LIN {X 0,Y 496.711,Z 403.86,A -85,B 0,C 180,E1 23580.115,E2 23580.115} C_VEL
LIN {X 0,Y 496.741,Z 403.852,A -85,B 0,C 180,E1 23576.65,E2 23576.65} C_VEL
LIN {X 0,Y 496.767,Z 403.854,A -85,B 0,C 180,E1 23573.18,E2 23573.18} C_VEL
LIN {X 0,Y 496.731,Z 403.861,A -85,B 0,C 180,E1 23569.68,E2 23569.68} C_VEL
LIN {X 0,Y 496.739,Z 403.856,A -85,B 0,C 180,E1 23566.141,E2 23566.141} C_VEL
LIN {X 0,Y 496.771,Z 403.853,A -85,B 0,C 180,E1 23562.669,E2 23562.669} C_VEL
LIN {X 0,Y 496.766,Z 403.847,A -85,B 0,C 180,E1 23559.041,E2 23559.041} C_VEL
LIN {X 0,Y 496.807,Z 404.124,A -85,B 0,C 180,E1 23556.819,E2 23556.819} C_VEL
LIN {X 0,Y 499.675,Z 411.051,A -85,B 0,C 180,E1 23555.782,E2 23555.782} C_VEL
LIN {X 0,Y 507.249,Z 429.235,A -85,B 0,C 180,E1 23553.293,E2 23553.293} C_VEL
LIN {X 0,Y 509.58,Z 435.728,A -85,B 0,C 180,E1 23552.475,E2 23552.475} C_VEL
LIN {X 0,Y 508.606,Z 453.094,A -85,B 0,C 180,E1 23551.014,E2 23551.014} C_VEL
LIN {X 0,Y 512.123,Z 472.591,A -85,B 0,C 180,E1 23550.372,E2 23550.372} C_VEL
LIN {X 0,Y 509.75,Z 617.433,A -85,B 0,C 180,E1 23548.089,E2 23548.089} C_VEL
LIN {X 0,Y 508.797,Z 625.124,A -85,B 0,C 180,E1 23548.03,E2 23548.03} C_VEL
LIN {X 0,Y 503.244,Z 645.629,A -85,B 0,C 180,E1 23548.096,E2 23548.096} C_VEL
LIN {X 0,Y 502.511,Z 652.229,A -85,B 0,C 180,E1 23548.038,E2 23548.038} C_VEL
LIN {X 0,Y 501.351,Z 717.097,A -85,B 0,C 180,E1 23546.975,E2 23546.975} C_VEL
LIN {X 0,Y 500.539,Z 738.052,A -85,B 0,C 180,E1 23546.417,E2 23546.417} C_VEL
LIN {X 0,Y 499.534,Z 757.461,A -85,B 0,C 180,E1 23545.684,E2 23545.684} C_VEL
LIN {X 0,Y 498.294,Z 776.687,A -85,B 0,C 180,E1 23544.746,E2 23544.746} C_VEL
LIN {X 0,Y 496.904,Z 795.621,A -85,B 0,C 180,E1 23543.587,E2 23543.587} C_VEL
LIN {X 0,Y 495.479,Z 813.178,A -85,B 0,C 180,E1 23542.277,E2 23542.277} C_VEL
LIN {X 0,Y 494.06,Z 829.63,A -85,B 0,C 180,E1 23540.808,E2 23540.808} C_VEL
LIN {X 0,Y 492.634,Z 845.536,A -85,B 0,C 180,E1 23539.11,E2 23539.11} C_VEL
LIN {X 0,Y 491.345,Z 860.076,A -85,B 0,C 180,E1 23537.269,E2 23537.269} C_VEL
LIN {X 0,Y 490.236,Z 873.347,A -85,B 0,C 180,E1 23535.28,E2 23535.28} C_VEL
LIN {X 0,Y 489.325,Z 886.414,A -85,B 0,C 180,E1 23532.986,E2 23532.986} C_VEL
LIN {X 0,Y 488.72,Z 897.123,A -85,B 0,C 180,E1 23530.736,E2 23530.736} C_VEL
LIN {X 0,Y 488.32,Z 905.885,A -85,B 0,C 180,E1 23528.491,E2 23528.491} C_VEL
LIN {X 0,Y 488.079,Z 913.183,A -85,B 0,C 180,E1 23526.152,E2 23526.152} C_VEL
LIN {X 0,Y 487.966,Z 918.575,A -85,B 0,C 180,E1 23523.868,E2 23523.868} C_VEL
LIN {X 0,Y 487.921,Z 922.481,A -85,B 0,C 180,E1 23521.499,E2 23521.499} C_VEL
LIN {X 0,Y 487.912,Z 924.811,A -85,B 0,C 180,E1 23519.053,E2 23519.053} C_VEL
LIN {X 0,Y 487.907,Z 925.448,A -85,B 0,C 180,E1 23516.662,E2 23516.662} C_VEL
LIN {X 0,Y 487.911,Z 924.503,A -85,B 0,C 180,E1 23514.321,E2 23514.321} C_VEL
LIN {X 0,Y 487.927,Z 921.952,A -85,B 0,C 180,E1 23512.021,E2 23512.021} C_VEL
LIN {X 0,Y 487.973,Z 917.691,A -85,B 0,C 180,E1 23509.632,E2 23509.632} C_VEL
LIN {X 0,Y 488.118,Z 911.798,A -85,B 0,C 180,E1 23507.275,E2 23507.275} C_VEL
LIN {X 0,Y 488.374,Z 904.684,A -85,B 0,C 180,E1 23505.068,E2 23505.068} C_VEL
LIN {X 0,Y 488.809,Z 895.342,A -85,B 0,C 180,E1 23502.76,E2 23502.76} C_VEL
LIN {X 0,Y 489.437,Z 884.661,A -85,B 0,C 180,E1 23500.592,E2 23500.592} C_VEL
LIN {X 0,Y 490.443,Z 870.664,A -85,B 0,C 180,E1 23498.202,E2 23498.202} C_VEL
LIN {X 0,Y 491.534,Z 857.477,A -85,B 0,C 180,E1 23496.304,E2 23496.304} C_VEL
LIN {X 0,Y 492.839,Z 842.493,A -85,B 0,C 180,E1 23494.477,E2 23494.477} C_VEL
LIN {X 0,Y 494.246,Z 826.553,A -85,B 0,C 180,E1 23492.838,E2 23492.838} C_VEL
LIN {X 0,Y 495.672,Z 809.764,A -85,B 0,C 180,E1 23491.385,E2 23491.385} C_VEL
LIN {X 0,Y 497.08,Z 792.089,A -85,B 0,C 180,E1 23490.113,E2 23490.113} C_VEL
LIN {X 0,Y 498.389,Z 773.462,A -85,B 0,C 180,E1 23489.02,E2 23489.02} C_VEL
LIN {X 0,Y 499.54,Z 754.515,A -85,B 0,C 180,E1 23488.134,E2 23488.134} C_VEL
LIN {X 0,Y 500.549,Z 733.899,A -85,B 0,C 180,E1 23487.4,E2 23487.4} C_VEL
LIN {X 0,Y 501.274,Z 713.46,A -85,B 0,C 180,E1 23486.893,E2 23486.893} C_VEL
LIN {X 0,Y 505.137,Z 479.595,A -85,B 0,C 180,E1 23483.179,E2 23483.179} C_VEL
LIN {X 0,Y 505.027,Z 471.969,A -85,B 0,C 180,E1 23483.036,E2 23483.036} C_VEL
LIN {X 0,Y 501.4,Z 452.019,A -85,B 0,C 180,E1 23482.346,E2 23482.346} C_VEL
LIN {X 0,Y 502.149,Z 437.999,A -85,B 0,C 180,E1 23481.121,E2 23481.121} C_VEL
LIN {X 0,Y 494.668,Z 418.979,A -85,B 0,C 180,E1 23478.615,E2 23478.615} C_VEL
LIN {X 0,Y 488.848,Z 405.013,A -85,B 0,C 180,E1 23476.605,E2 23476.605} C_VEL
LIN {X 0,Y 488.821,Z 404.811,A -85,B 0,C 180,E1 23472.99,E2 23472.99} C_VEL
LIN {X 0,Y 488.827,Z 404.843,A -85,B 0,C 180,E1 23469.4,E2 23469.4} C_VEL
LIN {X 0,Y 488.81,Z 404.825,A -85,B 0,C 180,E1 23465.825,E2 23465.825} C_VEL
LIN {X 0,Y 488.828,Z 404.838,A -85,B 0,C 180,E1 23462.333,E2 23462.333} C_VEL
LIN {X 0,Y 488.826,Z 404.833,A -85,B 0,C 180,E1 23458.697,E2 23458.697} C_VEL
LIN {X 0,Y 488.816,Z 404.833,A -85,B 0,C 180,E1 23455.109,E2 23455.109} C_VEL
LIN {X 0,Y 488.818,Z 404.835,A -85,B 0,C 180,E1 23451.549,E2 23451.549} C_VEL
LIN {X 0,Y 488.823,Z 404.846,A -85,B 0,C 180,E1 23448.019,E2 23448.019} C_VEL
LIN {X 0,Y 488.827,Z 404.84,A -85,B 0,C 180,E1 23444.39,E2 23444.39} C_VEL
LIN {X 0,Y 488.815,Z 404.84,A -85,B 0,C 180,E1 23440.813,E2 23440.813} C_VEL
LIN {X 0,Y 488.824,Z 404.834,A -85,B 0,C 180,E1 23437.262,E2 23437.262} C_VEL
LIN {X 0,Y 488.82,Z 404.845,A -85,B 0,C 180,E1 23433.642,E2 23433.642} C_VEL
LIN {X 0,Y 488.832,Z 404.835,A -85,B 0,C 180,E1 23430.075,E2 23430.075} C_VEL
LIN {X 0,Y 488.817,Z 404.83,A -85,B 0,C 180,E1 23426.482,E2 23426.482} C_VEL
LIN {X 0,Y 488.829,Z 404.846,A -85,B 0,C 180,E1 23422.87,E2 23422.87} C_VEL
LIN {X 0,Y 488.818,Z 404.831,A -85,B 0,C 180,E1 23419.228,E2 23419.228} C_VEL
LIN {X 0,Y 488.826,Z 404.834,A -85,B 0,C 180,E1 23415.664,E2 23415.664} C_VEL
LIN {X 0,Y 488.82,Z 404.846,A -85,B 0,C 180,E1 23412.043,E2 23412.043} C_VEL
LIN {X 0,Y 488.822,Z 404.831,A -85,B 0,C 180,E1 23408.469,E2 23408.469} C_VEL
LIN {X 0,Y 488.818,Z 404.841,A -85,B 0,C 180,E1 23404.811,E2 23404.811} C_VEL
LIN {X 0,Y 488.827,Z 404.84,A -85,B 0,C 180,E1 23401.172,E2 23401.172} C_VEL
LIN {X 0,Y 488.821,Z 404.834,A -85,B 0,C 180,E1 23397.538,E2 23397.538} C_VEL
LIN {X 0,Y 488.82,Z 404.843,A -85,B 0,C 180,E1 23394.012,E2 23394.012} C_VEL
LIN {X 0,Y 488.817,Z 404.843,A -85,B 0,C 180,E1 23390.345,E2 23390.345} C_VEL
LIN {X 0,Y 488.827,Z 404.84,A -85,B 0,C 180,E1 23386.757,E2 23386.757} C_VEL
LIN {X 0,Y 488.823,Z 404.836,A -85,B 0,C 180,E1 23383.115,E2 23383.115} C_VEL
LIN {X 0,Y 488.817,Z 404.839,A -85,B 0,C 180,E1 23379.527,E2 23379.527} C_VEL
LIN {X 0,Y 488.814,Z 404.842,A -85,B 0,C 180,E1 23375.852,E2 23375.852} C_VEL
LIN {X 0,Y 488.827,Z 404.839,A -85,B 0,C 180,E1 23372.335,E2 23372.335} C_VEL
LIN {X 0,Y 488.829,Z 404.839,A -85,B 0,C 180,E1 23368.699,E2 23368.699} C_VEL
LIN {X 0,Y 488.812,Z 404.84,A -85,B 0,C 180,E1 23365.111,E2 23365.111} C_VEL
LIN {X 0,Y 488.823,Z 404.841,A -85,B 0,C 180,E1 23361.552,E2 23361.552} C_VEL
LIN {X 0,Y 488.824,Z 404.846,A -85,B 0,C 180,E1 23358.021,E2 23358.021} C_VEL
LIN {X 0,Y 488.862,Z 405.087,A -85,B 0,C 180,E1 23355.482,E2 23355.482} C_VEL
LIN {X 0,Y 489.862,Z 407.901,A -85,B 0,C 180,E1 23355.072,E2 23355.072} C_VEL
LIN {X 0,Y 496.792,Z 422.284,A -85,B 0,C 180,E1 23353.182,E2 23353.182} C_VEL
LIN {X 0,Y 506.367,Z 443.634,A -85,B 0,C 180,E1 23350.626,E2 23350.626} C_VEL
LIN {X 0,Y 505.843,Z 455.638,A -85,B 0,C 180,E1 23349.815,E2 23349.815} C_VEL
LIN {X 0,Y 509.16,Z 477.639,A -85,B 0,C 180,E1 23349.149,E2 23349.149} C_VEL
LIN {X 0,Y 505.882,Z 697.396,A -85,B 0,C 180,E1 23345.689,E2 23345.689} C_VEL
LIN {X 0,Y 504.837,Z 762.385,A -85,B 0,C 180,E1 23344.65,E2 23344.65} C_VEL
LIN {X 0,Y 503.952,Z 783.667,A -85,B 0,C 180,E1 23344.113,E2 23344.113} C_VEL
LIN {X 0,Y 502.769,Z 806.1,A -85,B 0,C 180,E1 23343.331,E2 23343.331} C_VEL
LIN {X 0,Y 501.542,Z 826.208,A -85,B 0,C 180,E1 23342.432,E2 23342.432} C_VEL
LIN {X 0,Y 500.044,Z 845.015,A -85,B 0,C 180,E1 23341.373,E2 23341.373} C_VEL
LIN {X 0,Y 498.311,Z 865.469,A -85,B 0,C 180,E1 23339.976,E2 23339.976} C_VEL
LIN {X 0,Y 496.647,Z 883.732,A -85,B 0,C 180,E1 23338.5,E2 23338.5} C_VEL
LIN {X 0,Y 494.933,Z 901.867,A -85,B 0,C 180,E1 23336.758,E2 23336.758} C_VEL
LIN {X 0,Y 493.329,Z 918.653,A -85,B 0,C 180,E1 23334.871,E2 23334.871} C_VEL
LIN {X 0,Y 491.921,Z 934.162,A -85,B 0,C 180,E1 23332.846,E2 23332.846} C_VEL
LIN {X 0,Y 490.71,Z 948.618,A -85,B 0,C 180,E1 23330.642,E2 23330.642} C_VEL
LIN {X 0,Y 489.723,Z 961.442,A -85,B 0,C 180,E1 23328.328,E2 23328.328} C_VEL
LIN {X 0,Y 488.985,Z 972.802,A -85,B 0,C 180,E1 23325.904,E2 23325.904} C_VEL
LIN {X 0,Y 488.492,Z 982.252,A -85,B 0,C 180,E1 23323.496,E2 23323.496} C_VEL
LIN {X 0,Y 488.184,Z 989.875,A -85,B 0,C 180,E1 23321.102,E2 23321.102} C_VEL
LIN {X 0,Y 488.014,Z 996.141,A -85,B 0,C 180,E1 23318.604,E2 23318.604} C_VEL
LIN {X 0,Y 487.94,Z 1000.819,A -85,B 0,C 180,E1 23316.119,E2 23316.119} C_VEL
LIN {X 0,Y 487.912,Z 1003.791,A -85,B 0,C 180,E1 23313.639,E2 23313.639} C_VEL
LIN {X 0,Y 487.908,Z 1005.304,A -85,B 0,C 180,E1 23311.059,E2 23311.059} C_VEL
LIN {X 0,Y 487.907,Z 1005.259,A -85,B 0,C 180,E1 23308.711,E2 23308.711} C_VEL
LIN {X 0,Y 487.91,Z 1003.674,A -85,B 0,C 180,E1 23306.243,E2 23306.243} C_VEL
LIN {X 0,Y 487.944,Z 1000.637,A -85,B 0,C 180,E1 23303.768,E2 23303.768} C_VEL
LIN {X 0,Y 488.018,Z 995.896,A -85,B 0,C 180,E1 23301.282,E2 23301.282} C_VEL
LIN {X 0,Y 488.206,Z 989.183,A -85,B 0,C 180,E1 23298.664,E2 23298.664} C_VEL
LIN {X 0,Y 488.532,Z 981.438,A -85,B 0,C 180,E1 23296.269,E2 23296.269} C_VEL
LIN {X 0,Y 489.045,Z 971.794,A -85,B 0,C 180,E1 23293.859,E2 23293.859} C_VEL
LIN {X 0,Y 489.807,Z 960.2,A -85,B 0,C 180,E1 23291.434,E2 23291.434} C_VEL
LIN {X 0,Y 490.765,Z 947.883,A -85,B 0,C 180,E1 23289.241,E2 23289.241} C_VEL
LIN {X 0,Y 491.917,Z 934.198,A -85,B 0,C 180,E1 23287.16,E2 23287.16} C_VEL
LIN {X 0,Y 493.326,Z 918.696,A -85,B 0,C 180,E1 23285.134,E2 23285.134} C_VEL
LIN {X 0,Y 494.944,Z 901.731,A -85,B 0,C 180,E1 23283.228,E2 23283.228} C_VEL
LIN {X 0,Y 496.642,Z 883.791,A -85,B 0,C 180,E1 23281.505,E2 23281.505} C_VEL
LIN {X 0,Y 498.306,Z 865.543,A -85,B 0,C 180,E1 23280.029,E2 23280.029} C_VEL
LIN {X 0,Y 500.043,Z 845.02,A -85,B 0,C 180,E1 23278.627,E2 23278.627} C_VEL
LIN {X 0,Y 501.533,Z 826.304,A -85,B 0,C 180,E1 23277.573,E2 23277.573} C_VEL
LIN {X 0,Y 502.801,Z 805.216,A -85,B 0,C 180,E1 23276.636,E2 23276.636} C_VEL
LIN {X 0,Y 503.96,Z 782.783,A -85,B 0,C 180,E1 23275.868,E2 23275.868} C_VEL
LIN {X 0,Y 504.819,Z 761.32,A -85,B 0,C 180,E1 23275.337,E2 23275.337} C_VEL
LIN {X 0,Y 506.726,Z 630.415,A -85,B 0,C 180,E1 23273.284,E2 23273.284} C_VEL
LIN {X 0,Y 508.834,Z 475.555,A -85,B 0,C 180,E1 23270.839,E2 23270.839} C_VEL
LIN {X 0,Y 505.533,Z 454.855,A -85,B 0,C 180,E1 23270.2,E2 23270.2} C_VEL
LIN {X 0,Y 506.097,Z 443.386,A -85,B 0,C 180,E1 23269.404,E2 23269.404} C_VEL
LIN {X 0,Y 495.503,Z 419.708,A -85,B 0,C 180,E1 23266.588,E2 23266.588} C_VEL
LIN {X 0,Y 490.039,Z 408.23,A -85,B 0,C 180,E1 23265.072,E2 23265.072} C_VEL
LIN {X 0,Y 488.851,Z 405.059,A -85,B 0,C 180,E1 23264.596,E2 23264.596} C_VEL
LIN {X 0,Y 488.793,Z 404.851,A -85,B 0,C 180,E1 23261.175,E2 23261.175} C_VEL
LIN {X 0,Y 488.817,Z 404.848,A -85,B 0,C 180,E1 23257.672,E2 23257.672} C_VEL
LIN {X 0,Y 488.825,Z 404.842,A -85,B 0,C 180,E1 23254.086,E2 23254.086} C_VEL
LIN {X 0,Y 488.781,Z 404.849,A -85,B 0,C 180,E1 23250.621,E2 23250.621} C_VEL
LIN {X 0,Y 488.772,Z 404.844,A -85,B 0,C 180,E1 23247.009,E2 23247.009} C_VEL
LIN {X 0,Y 488.826,Z 404.841,A -85,B 0,C 180,E1 23243.612,E2 23243.612} C_VEL
LIN {X 0,Y 488.769,Z 404.846,A -85,B 0,C 180,E1 23240.225,E2 23240.225} C_VEL
LIN {X 0,Y 488.751,Z 404.852,A -85,B 0,C 180,E1 23236.642,E2 23236.642} C_VEL
LIN {X 0,Y 488.795,Z 404.851,A -85,B 0,C 180,E1 23233.244,E2 23233.244} C_VEL
LIN {X 0,Y 488.782,Z 404.851,A -85,B 0,C 180,E1 23229.775,E2 23229.775} C_VEL
LIN {X 0,Y 488.76,Z 404.85,A -85,B 0,C 180,E1 23226.342,E2 23226.342} C_VEL
LIN {X 0,Y 488.806,Z 404.843,A -85,B 0,C 180,E1 23222.931,E2 23222.931} C_VEL
LIN {X 0,Y 488.801,Z 404.846,A -85,B 0,C 180,E1 23219.531,E2 23219.531} C_VEL
LIN {X 0,Y 488.778,Z 404.842,A -85,B 0,C 180,E1 23216.011,E2 23216.011} C_VEL
LIN {X 0,Y 488.804,Z 404.847,A -85,B 0,C 180,E1 23212.477,E2 23212.477} C_VEL
LIN {X 0,Y 488.833,Z 404.841,A -85,B 0,C 180,E1 23208.915,E2 23208.915} C_VEL
LIN {X 0,Y 488.813,Z 404.849,A -85,B 0,C 180,E1 23205.307,E2 23205.307} C_VEL
LIN {X 0,Y 488.8,Z 404.848,A -85,B 0,C 180,E1 23201.761,E2 23201.761} C_VEL
LIN {X 0,Y 488.826,Z 404.827,A -85,B 0,C 180,E1 23198.21,E2 23198.21} C_VEL
LIN {X 0,Y 488.87,Z 405.268,A -85,B 0,C 180,E1 23197.562,E2 23197.562} C_VEL
LIN {X 0,Y 496.721,Z 423.489,A -85,B 0,C 180,E1 23194.866,E2 23194.866} C_VEL
LIN {X 0,Y 502.751,Z 438.85,A -85,B 0,C 180,E1 23192.811,E2 23192.811} C_VEL
LIN {X 0,Y 501.912,Z 453.11,A -85,B 0,C 180,E1 23191.6,E2 23191.6} C_VEL
LIN {X 0,Y 505.677,Z 473.944,A -85,B 0,C 180,E1 23190.891,E2 23190.891} C_VEL
LIN {X 0,Y 502.511,Z 652.229,A -85,B 0,C 180,E1 23188.038,E2 23188.038} C_VEL
LIN {X 0,Y 501.556,Z 659.917,A -85,B 0,C 180,E1 23187.978,E2 23187.978} C_VEL
LIN {X 0,Y 495.97,Z 680.411,A -85,B 0,C 180,E1 23188.046,E2 23188.046} C_VEL
LIN {X 0,Y 495.215,Z 687.011,A -85,B 0,C 180,E1 23187.989,E2 23187.989} C_VEL
LIN {X 0,Y 494.51,Z 719.382,A -85,B 0,C 180,E1 23187.421,E2 23187.421} C_VEL
LIN {X 0,Y 493.662,Z 739.881,A -85,B 0,C 180,E1 23186.854,E2 23186.854} C_VEL
LIN {X 0,Y 492.59,Z 759.03,A -85,B 0,C 180,E1 23186.111,E2 23186.111} C_VEL
LIN {X 0,Y 491.254,Z 778.214,A -85,B 0,C 180,E1 23185.151,E2 23185.151} C_VEL
LIN {X 0,Y 489.725,Z 797.454,A -85,B 0,C 180,E1 23183.943,E2 23183.943} C_VEL
LIN {X 0,Y 488.108,Z 815.828,A -85,B 0,C 180,E1 23182.527,E2 23182.527} C_VEL
LIN {X 0,Y 486.591,Z 831.937,A -85,B 0,C 180,E1 23181.04,E2 23181.04} C_VEL
LIN {X 0,Y 485.097,Z 847.586,A -85,B 0,C 180,E1 23179.326,E2 23179.326} C_VEL
LIN {X 0,Y 483.669,Z 862.482,A -85,B 0,C 180,E1 23177.381,E2 23177.381} C_VEL
LIN {X 0,Y 482.491,Z 875.405,A -85,B 0,C 180,E1 23175.371,E2 23175.371} C_VEL
LIN {X 0,Y 481.52,Z 887.09,A -85,B 0,C 180,E1 23173.21,E2 23173.21} C_VEL
LIN {X 0,Y 480.801,Z 897.389,A -85,B 0,C 180,E1 23170.92,E2 23170.92} C_VEL
LIN {X 0,Y 480.336,Z 906.546,A -85,B 0,C 180,E1 23168.486,E2 23168.486} C_VEL
LIN {X 0,Y 480.083,Z 913.675,A -85,B 0,C 180,E1 23166.11,E2 23166.11} C_VEL
LIN {X 0,Y 479.968,Z 919.002,A -85,B 0,C 180,E1 23163.778,E2 23163.778} C_VEL
LIN {X 0,Y 479.921,Z 922.809,A -85,B 0,C 180,E1 23161.329,E2 23161.329} C_VEL
LIN {X 0,Y 479.916,Z 924.888,A -85,B 0,C 180,E1 23158.951,E2 23158.951} C_VEL
LIN {X 0,Y 479.904,Z 925.413,A -85,B 0,C 180,E1 23156.475,E2 23156.475} C_VEL
LIN {X 0,Y 479.911,Z 924.355,A -85,B 0,C 180,E1 23154.098,E2 23154.098} C_VEL
LIN {X 0,Y 479.921,Z 921.621,A -85,B 0,C 180,E1 23151.69,E2 23151.69} C_VEL
LIN {X 0,Y 479.993,Z 917.308,A -85,B 0,C 180,E1 23149.328,E2 23149.328} C_VEL
LIN {X 0,Y 480.157,Z 911.311,A -85,B 0,C 180,E1 23146.946,E2 23146.946} C_VEL
LIN {X 0,Y 480.464,Z 903.7,A -85,B 0,C 180,E1 23144.606,E2 23144.606} C_VEL
LIN {X 0,Y 481.038,Z 893.677,A -85,B 0,C 180,E1 23142.115,E2 23142.115} C_VEL
LIN {X 0,Y 481.831,Z 883.067,A -85,B 0,C 180,E1 23139.915,E2 23139.915} C_VEL
LIN {X 0,Y 482.9,Z 870.365,A -85,B 0,C 180,E1 23137.732,E2 23137.732} C_VEL
LIN {X 0,Y 484.206,Z 856.1,A -85,B 0,C 180,E1 23135.686,E2 23135.686} C_VEL
LIN {X 0,Y 485.591,Z 841.256,A -85,B 0,C 180,E1 23133.894,E2 23133.894} C_VEL
LIN {X 0,Y 487.137,Z 824.939,A -85,B 0,C 180,E1 23132.232,E2 23132.232} C_VEL
LIN {X 0,Y 488.769,Z 806.901,A -85,B 0,C 180,E1 23130.701,E2 23130.701} C_VEL
LIN {X 0,Y 490.227,Z 789.454,A -85,B 0,C 180,E1 23129.472,E2 23129.472} C_VEL
LIN {X 0,Y 491.612,Z 771.326,A -85,B 0,C 180,E1 23128.424,E2 23128.424} C_VEL
LIN {X 0,Y 492.816,Z 751.622,A -85,B 0,C 180,E1 23127.527,E2 23127.527} C_VEL
LIN {X 0,Y 493.826,Z 731.788,A -85,B 0,C 180,E1 23126.849,E2 23126.849} C_VEL
LIN {X 0,Y 494.543,Z 710.498,A -85,B 0,C 180,E1 23126.346,E2 23126.346} C_VEL
LIN {X 0,Y 498.752,Z 474.593,A -85,B 0,C 180,E1 23122.554,E2 23122.554} C_VEL
LIN {X 0,Y 494.672,Z 452.27,A -85,B 0,C 180,E1 23121.776,E2 23121.776} C_VEL
LIN {X 0,Y 495.272,Z 441.414,A -85,B 0,C 180,E1 23120.821,E2 23120.821} C_VEL
LIN {X 0,Y 488.004,Z 422.954,A -85,B 0,C 180,E1 23118.341,E2 23118.341} C_VEL
LIN {X 0,Y 481.996,Z 409.011,A -85,B 0,C 180,E1 23116.319,E2 23116.319} C_VEL
LIN {X 0,Y 480.894,Z 405.949,A -85,B 0,C 180,E1 23115.816,E2 23115.816} C_VEL
LIN {X 0,Y 480.869,Z 405.8,A -85,B 0,C 180,E1 23112.2,E2 23112.2} C_VEL
LIN {X 0,Y 480.887,Z 405.809,A -85,B 0,C 180,E1 23108.661,E2 23108.661} C_VEL
LIN {X 0,Y 480.889,Z 405.828,A -85,B 0,C 180,E1 23105.031,E2 23105.031} C_VEL
LIN {X 0,Y 480.878,Z 405.834,A -85,B 0,C 180,E1 23101.429,E2 23101.429} C_VEL
LIN {X 0,Y 480.881,Z 405.834,A -85,B 0,C 180,E1 23097.806,E2 23097.806} C_VEL
LIN {X 0,Y 480.886,Z 405.825,A -85,B 0,C 180,E1 23094.183,E2 23094.183} C_VEL
LIN {X 0,Y 480.888,Z 405.819,A -85,B 0,C 180,E1 23090.479,E2 23090.479} C_VEL
LIN {X 0,Y 480.875,Z 405.82,A -85,B 0,C 180,E1 23086.999,E2 23086.999} C_VEL
LIN {X 0,Y 480.882,Z 405.83,A -85,B 0,C 180,E1 23083.326,E2 23083.326} C_VEL
LIN {X 0,Y 480.885,Z 405.831,A -85,B 0,C 180,E1 23079.707,E2 23079.707} C_VEL
LIN {X 0,Y 480.884,Z 405.819,A -85,B 0,C 180,E1 23076.018,E2 23076.018} C_VEL
LIN {X 0,Y 480.881,Z 405.824,A -85,B 0,C 180,E1 23072.416,E2 23072.416} C_VEL
LIN {X 0,Y 480.881,Z 405.835,A -85,B 0,C 180,E1 23068.705,E2 23068.705} C_VEL
LIN {X 0,Y 480.882,Z 405.818,A -85,B 0,C 180,E1 23065.098,E2 23065.098} C_VEL
LIN {X 0,Y 480.885,Z 405.827,A -85,B 0,C 180,E1 23061.466,E2 23061.466} C_VEL
LIN {X 0,Y 480.884,Z 405.83,A -85,B 0,C 180,E1 23057.797,E2 23057.797} C_VEL
LIN {X 0,Y 480.881,Z 405.821,A -85,B 0,C 180,E1 23054.203,E2 23054.203} C_VEL
LIN {X 0,Y 480.885,Z 405.833,A -85,B 0,C 180,E1 23050.543,E2 23050.543} C_VEL
LIN {X 0,Y 480.881,Z 405.827,A -85,B 0,C 180,E1 23046.927,E2 23046.927} C_VEL
LIN {X 0,Y 480.883,Z 405.814,A -85,B 0,C 180,E1 23043.338,E2 23043.338} C_VEL
LIN {X 0,Y 480.883,Z 405.828,A -85,B 0,C 180,E1 23039.643,E2 23039.643} C_VEL
LIN {X 0,Y 480.88,Z 405.83,A -85,B 0,C 180,E1 23036.066,E2 23036.066} C_VEL
LIN {X 0,Y 480.879,Z 405.816,A -85,B 0,C 180,E1 23032.473,E2 23032.473} C_VEL
LIN {X 0,Y 480.885,Z 405.824,A -85,B 0,C 180,E1 23028.851,E2 23028.851} C_VEL
LIN {X 0,Y 480.887,Z 405.833,A -85,B 0,C 180,E1 23025.183,E2 23025.183} C_VEL
LIN {X 0,Y 480.88,Z 405.832,A -85,B 0,C 180,E1 23021.577,E2 23021.577} C_VEL
LIN {X 0,Y 480.875,Z 405.829,A -85,B 0,C 180,E1 23017.893,E2 23017.893} C_VEL
LIN {X 0,Y 480.888,Z 405.829,A -85,B 0,C 180,E1 23014.376,E2 23014.376} C_VEL
LIN {X 0,Y 480.891,Z 405.828,A -85,B 0,C 180,E1 23010.751,E2 23010.751} C_VEL
LIN {X 0,Y 480.874,Z 405.83,A -85,B 0,C 180,E1 23007.134,E2 23007.134} C_VEL
LIN {X 0,Y 480.878,Z 405.835,A -85,B 0,C 180,E1 23003.512,E2 23003.512} C_VEL
LIN {X 0,Y 480.89,Z 405.826,A -85,B 0,C 180,E1 22999.869,E2 22999.869} C_VEL
LIN {X 0,Y 480.919,Z 406.048,A -85,B 0,C 180,E1 22996.314,E2 22996.314} C_VEL
LIN {X 0,Y 481.823,Z 408.683,A -85,B 0,C 180,E1 22995.892,E2 22995.892} C_VEL
LIN {X 0,Y 487.309,Z 419.889,A -85,B 0,C 180,E1 22994.353,E2 22994.353} C_VEL
LIN {X 0,Y 495.136,Z 437.007,A -85,B 0,C 180,E1 22992.175,E2 22992.175} C_VEL
LIN {X 0,Y 499.613,Z 447.338,A -85,B 0,C 180,E1 22990.953,E2 22990.953} C_VEL
LIN {X 0,Y 499.254,Z 455.651,A -85,B 0,C 180,E1 22990.396,E2 22990.396} C_VEL
LIN {X 0,Y 502.726,Z 479.022,A -85,B 0,C 180,E1 22989.673,E2 22989.673} C_VEL
LIN {X 0,Y 499.168,Z 698.972,A -85,B 0,C 180,E1 22986.168,E2 22986.168} C_VEL
LIN {X 0,Y 498.066,Z 762.045,A -85,B 0,C 180,E1 22985.147,E2 22985.147} C_VEL
LIN {X 0,Y 497.129,Z 783.164,A -85,B 0,C 180,E1 22984.608,E2 22984.608} C_VEL
LIN {X 0,Y 495.848,Z 805.634,A -85,B 0,C 180,E1 22983.819,E2 22983.819} C_VEL
LIN {X 0,Y 494.485,Z 826.231,A -85,B 0,C 180,E1 22982.884,E2 22982.884} C_VEL
LIN {X 0,Y 492.886,Z 845.938,A -85,B 0,C 180,E1 22981.772,E2 22981.772} C_VEL
LIN {X 0,Y 491.157,Z 866.165,A -85,B 0,C 180,E1 22980.395,E2 22980.395} C_VEL
LIN {X 0,Y 489.457,Z 883.73,A -85,B 0,C 180,E1 22978.958,E2 22978.958} C_VEL
LIN {X 0,Y 487.609,Z 901.678,A -85,B 0,C 180,E1 22977.213,E2 22977.213} C_VEL
LIN {X 0,Y 485.854,Z 918.652,A -85,B 0,C 180,E1 22975.281,E2 22975.281} C_VEL
LIN {X 0,Y 484.328,Z 934.161,A -85,B 0,C 180,E1 22973.225,E2 22973.225} C_VEL
LIN {X 0,Y 482.999,Z 948.617,A -85,B 0,C 180,E1 22970.987,E2 22970.987} C_VEL
LIN {X 0,Y 481.959,Z 960.805,A -85,B 0,C 180,E1 22968.759,E2 22968.759} C_VEL
LIN {X 0,Y 481.117,Z 972.538,A -85,B 0,C 180,E1 22966.235,E2 22966.235} C_VEL
LIN {X 0,Y 480.579,Z 981.845,A -85,B 0,C 180,E1 22963.845,E2 22963.845} C_VEL
LIN {X 0,Y 480.228,Z 989.522,A -85,B 0,C 180,E1 22961.41,E2 22961.41} C_VEL
LIN {X 0,Y 480.024,Z 996.141,A -85,B 0,C 180,E1 22958.748,E2 22958.748} C_VEL
LIN {X 0,Y 479.944,Z 1000.819,A -85,B 0,C 180,E1 22956.221,E2 22956.221} C_VEL
LIN {X 0,Y 479.912,Z 1003.82,A -85,B 0,C 180,E1 22953.668,E2 22953.668} C_VEL
LIN {X 0,Y 479.908,Z 1005.304,A -85,B 0,C 180,E1 22951.077,E2 22951.077} C_VEL
LIN {X 0,Y 479.906,Z 1005.259,A -85,B 0,C 180,E1 22948.689,E2 22948.689} C_VEL
LIN {X 0,Y 479.911,Z 1003.673,A -85,B 0,C 180,E1 22946.18,E2 22946.18} C_VEL
LIN {X 0,Y 479.949,Z 1000.637,A -85,B 0,C 180,E1 22943.664,E2 22943.664} C_VEL
LIN {X 0,Y 480.029,Z 995.896,A -85,B 0,C 180,E1 22941.136,E2 22941.136} C_VEL
LIN {X 0,Y 480.239,Z 989.182,A -85,B 0,C 180,E1 22938.473,E2 22938.473} C_VEL
LIN {X 0,Y 480.598,Z 981.437,A -85,B 0,C 180,E1 22936.038,E2 22936.038} C_VEL
LIN {X 0,Y 481.16,Z 971.793,A -85,B 0,C 180,E1 22933.587,E2 22933.587} C_VEL
LIN {X 0,Y 482.005,Z 960.198,A -85,B 0,C 180,E1 22931.122,E2 22931.122} C_VEL
LIN {X 0,Y 483.059,Z 947.882,A -85,B 0,C 180,E1 22928.894,E2 22928.894} C_VEL
LIN {X 0,Y 484.371,Z 933.78,A -85,B 0,C 180,E1 22926.72,E2 22926.72} C_VEL
LIN {X 0,Y 485.902,Z 918.189,A -85,B 0,C 180,E1 22924.662,E2 22924.662} C_VEL
LIN {X 0,Y 487.637,Z 901.386,A -85,B 0,C 180,E1 22922.757,E2 22922.757} C_VEL
LIN {X 0,Y 489.452,Z 883.789,A -85,B 0,C 180,E1 22921.047,E2 22921.047} C_VEL
LIN {X 0,Y 491.159,Z 866.168,A -85,B 0,C 180,E1 22919.605,E2 22919.605} C_VEL
LIN {X 0,Y 492.903,Z 845.473,A -85,B 0,C 180,E1 22918.205,E2 22918.205} C_VEL
LIN {X 0,Y 494.538,Z 824.894,A -85,B 0,C 180,E1 22917.057,E2 22917.057} C_VEL
LIN {X 0,Y 495.912,Z 803.759,A -85,B 0,C 180,E1 22916.118,E2 22916.118} C_VEL
LIN {X 0,Y 497.116,Z 781.867,A -85,B 0,C 180,E1 22915.369,E2 22915.369} C_VEL
LIN {X 0,Y 498.015,Z 760.541,A -85,B 0,C 180,E1 22914.84,E2 22914.84} C_VEL
LIN {X 0,Y 500.658,Z 591.901,A -85,B 0,C 180,E1 22912.17,E2 22912.17} C_VEL
LIN {X 0,Y 502.311,Z 476.728,A -85,B 0,C 180,E1 22910.316,E2 22910.316} C_VEL
LIN {X 0,Y 498.895,Z 454.426,A -85,B 0,C 180,E1 22909.603,E2 22909.603} C_VEL
LIN {X 0,Y 499.207,Z 446.537,A -85,B 0,C 180,E1 22909.033,E2 22909.033} C_VEL
LIN {X 0,Y 488.88,Z 423.411,A -85,B 0,C 180,E1 22906.216,E2 22906.216} C_VEL
LIN {X 0,Y 482.281,Z 409.446,A -85,B 0,C 180,E1 22904.319,E2 22904.319} C_VEL
LIN {X 0,Y 480.913,Z 406.047,A -85,B 0,C 180,E1 22903.783,E2 22903.783} C_VEL
LIN {X 0,Y 480.897,Z 405.83,A -85,B 0,C 180,E1 22900.272,E2 22900.272} C_VEL
LIN {X 0,Y 480.85,Z 405.837,A -85,B 0,C 180,E1 22896.788,E2 22896.788} C_VEL
LIN {X 0,Y 480.845,Z 405.84,A -85,B 0,C 180,E1 22893.079,E2 22893.079} C_VEL
LIN {X 0,Y 480.885,Z 405.831,A -85,B 0,C 180,E1 22889.653,E2 22889.653} C_VEL
LIN {X 0,Y 480.855,Z 405.831,A -85,B 0,C 180,E1 22886.156,E2 22886.156} C_VEL
LIN {X 0,Y 480.824,Z 405.84,A -85,B 0,C 180,E1 22882.754,E2 22882.754} C_VEL
LIN {X 0,Y 480.852,Z 405.839,A -85,B 0,C 180,E1 22879.274,E2 22879.274} C_VEL
LIN {X 0,Y 480.849,Z 405.841,A -85,B 0,C 180,E1 22875.807,E2 22875.807} C_VEL
LIN {X 0,Y 480.811,Z 405.84,A -85,B 0,C 180,E1 22872.368,E2 22872.368} C_VEL
LIN {X 0,Y 480.836,Z 405.832,A -85,B 0,C 180,E1 22868.851,E2 22868.851} C_VEL
LIN {X 0,Y 480.868,Z 405.832,A -85,B 0,C 180,E1 22865.488,E2 22865.488} C_VEL
LIN {X 0,Y 480.831,Z 405.833,A -85,B 0,C 180,E1 22862.026,E2 22862.026} C_VEL
LIN {X 0,Y 480.845,Z 405.836,A -85,B 0,C 180,E1 22858.451,E2 22858.451} C_VEL
LIN {X 0,Y 480.892,Z 405.836,A -85,B 0,C 180,E1 22854.99,E2 22854.99} C_VEL
LIN {X 0,Y 480.861,Z 405.836,A -85,B 0,C 180,E1 22851.51,E2 22851.51} C_VEL
LIN {X 0,Y 480.854,Z 405.836,A -85,B 0,C 180,E1 22847.998,E2 22847.998} C_VEL
LIN {X 0,Y 480.889,Z 405.83,A -85,B 0,C 180,E1 22844.442,E2 22844.442} C_VEL
LIN {X 0,Y 480.893,Z 405.831,A -85,B 0,C 180,E1 22840.821,E2 22840.821} C_VEL
LIN {X 0,Y 480.928,Z 406.072,A -85,B 0,C 180,E1 22838.423,E2 22838.423} C_VEL
LIN {X 0,Y 483.955,Z 413.206,A -85,B 0,C 180,E1 22837.272,E2 22837.272} C_VEL
LIN {X 0,Y 490.749,Z 429.077,A -85,B 0,C 180,E1 22834.926,E2 22834.926} C_VEL
LIN {X 0,Y 495.93,Z 442.4,A -85,B 0,C 180,E1 22833.12,E2 22833.12} C_VEL
LIN {X 0,Y 495.272,Z 453.159,A -85,B 0,C 180,E1 22832.202,E2 22832.202} C_VEL
LIN {X 0,Y 499.279,Z 475.412,A -85,B 0,C 180,E1 22831.423,E2 22831.423} C_VEL
LIN {X 0,Y 495.215,Z 687.011,A -85,B 0,C 180,E1 22827.989,E2 22827.989} C_VEL
LIN {X 0,Y 494.246,Z 694.703,A -85,B 0,C 180,E1 22827.931,E2 22827.931} C_VEL
LIN {X 0,Y 488.543,Z 715.162,A -85,B 0,C 180,E1 22827.981,E2 22827.981} C_VEL
LIN {X 0,Y 487.697,Z 721.698,A -85,B 0,C 180,E1 22827.879,E2 22827.879} C_VEL
LIN {X 0,Y 486.787,Z 741.911,A -85,B 0,C 180,E1 22827.293,E2 22827.293} C_VEL
LIN {X 0,Y 485.597,Z 761.845,A -85,B 0,C 180,E1 22826.495,E2 22826.495} C_VEL
LIN {X 0,Y 484.137,Z 781.219,A -85,B 0,C 180,E1 22825.483,E2 22825.483} C_VEL
LIN {X 0,Y 482.562,Z 799.332,A -85,B 0,C 180,E1 22824.306,E2 22824.306} C_VEL
LIN {X 0,Y 480.892,Z 816.947,A -85,B 0,C 180,E1 22822.917,E2 22822.917} C_VEL
LIN {X 0,Y 479.206,Z 833.543,A -85,B 0,C 180,E1 22821.351,E2 22821.351} C_VEL
LIN {X 0,Y 477.628,Z 848.877,A -85,B 0,C 180,E1 22819.634,E2 22819.634} C_VEL
LIN {X 0,Y 476.099,Z 863.701,A -85,B 0,C 180,E1 22817.661,E2 22817.661} C_VEL
LIN {X 0,Y 474.787,Z 876.976,A -85,B 0,C 180,E1 22815.548,E2 22815.548} C_VEL
LIN {X 0,Y 473.773,Z 888.039,A -85,B 0,C 180,E1 22813.449,E2 22813.449} C_VEL
LIN {X 0,Y 472.991,Z 898.003,A -85,B 0,C 180,E1 22811.188,E2 22811.188} C_VEL
LIN {X 0,Y 472.443,Z 906.654,A -85,B 0,C 180,E1 22808.783,E2 22808.783} C_VEL
LIN {X 0,Y 472.117,Z 913.556,A -85,B 0,C 180,E1 22806.365,E2 22806.365} C_VEL
LIN {X 0,Y 471.967,Z 919.448,A -85,B 0,C 180,E1 22803.636,E2 22803.636} C_VEL
LIN {X 0,Y 471.923,Z 923.167,A -85,B 0,C 180,E1 22801.124,E2 22801.124} C_VEL
LIN {X 0,Y 471.909,Z 925.048,A -85,B 0,C 180,E1 22798.697,E2 22798.697} C_VEL
LIN {X 0,Y 471.906,Z 925.378,A -85,B 0,C 180,E1 22796.28,E2 22796.28} C_VEL
LIN {X 0,Y 471.908,Z 924.185,A -85,B 0,C 180,E1 22793.868,E2 22793.868} C_VEL
LIN {X 0,Y 471.928,Z 921.486,A -85,B 0,C 180,E1 22791.498,E2 22791.498} C_VEL
LIN {X 0,Y 472.018,Z 916.993,A -85,B 0,C 180,E1 22789.036,E2 22789.036} C_VEL
LIN {X 0,Y 472.231,Z 910.689,A -85,B 0,C 180,E1 22786.479,E2 22786.479} C_VEL
LIN {X 0,Y 472.648,Z 903.049,A -85,B 0,C 180,E1 22784.077,E2 22784.077} C_VEL
LIN {X 0,Y 473.292,Z 893.625,A -85,B 0,C 180,E1 22781.698,E2 22781.698} C_VEL
LIN {X 0,Y 474.19,Z 882.858,A -85,B 0,C 180,E1 22779.463,E2 22779.463} C_VEL
LIN {X 0,Y 475.311,Z 870.804,A -85,B 0,C 180,E1 22777.37,E2 22777.37} C_VEL
LIN {X 0,Y 476.638,Z 857.377,A -85,B 0,C 180,E1 22775.414,E2 22775.414} C_VEL
LIN {X 0,Y 478.124,Z 842.648,A -85,B 0,C 180,E1 22773.594,E2 22773.594} C_VEL
LIN {X 0,Y 479.813,Z 826.079,A -85,B 0,C 180,E1 22771.871,E2 22771.871} C_VEL
LIN {X 0,Y 481.517,Z 808.615,A -85,B 0,C 180,E1 22770.354,E2 22770.354} C_VEL
LIN {X 0,Y 483.074,Z 791.417,A -85,B 0,C 180,E1 22769.108,E2 22769.108} C_VEL
LIN {X 0,Y 484.613,Z 772.414,A -85,B 0,C 180,E1 22767.988,E2 22767.988} C_VEL
LIN {X 0,Y 485.896,Z 752.864,A -85,B 0,C 180,E1 22767.078,E2 22767.078} C_VEL
LIN {X 0,Y 486.99,Z 732.845,A -85,B 0,C 180,E1 22766.378,E2 22766.378} C_VEL
LIN {X 0,Y 487.769,Z 711.561,A -85,B 0,C 180,E1 22765.861,E2 22765.861} C_VEL
LIN {X 0,Y 492.291,Z 475.937,A -85,B 0,C 180,E1 22762.019,E2 22762.019} C_VEL
LIN {X 0,Y 487.987,Z 452.053,A -85,B 0,C 180,E1 22761.158,E2 22761.158} C_VEL
LIN {X 0,Y 488.41,Z 444.838,A -85,B 0,C 180,E1 22760.512,E2 22760.512} C_VEL
LIN {X 0,Y 480.747,Z 425.236,A -85,B 0,C 180,E1 22757.826,E2 22757.826} C_VEL
LIN {X 0,Y 473.996,Z 409.876,A -85,B 0,C 180,E1 22755.519,E2 22755.519} C_VEL
LIN {X 0,Y 472.969,Z 406.967,A -85,B 0,C 180,E1 22755.04,E2 22755.04} C_VEL
LIN {X 0,Y 472.942,Z 406.795,A -85,B 0,C 180,E1 22751.509,E2 22751.509} C_VEL
LIN {X 0,Y 472.93,Z 406.783,A -85,B 0,C 180,E1 22747.892,E2 22747.892} C_VEL
LIN {X 0,Y 472.95,Z 406.826,A -85,B 0,C 180,E1 22744.238,E2 22744.238} C_VEL
LIN {X 0,Y 472.948,Z 406.824,A -85,B 0,C 180,E1 22740.577,E2 22740.577} C_VEL
LIN {X 0,Y 472.95,Z 406.821,A -85,B 0,C 180,E1 22736.944,E2 22736.944} C_VEL
LIN {X 0,Y 472.937,Z 406.823,A -85,B 0,C 180,E1 22733.25,E2 22733.25} C_VEL
LIN {X 0,Y 472.945,Z 406.821,A -85,B 0,C 180,E1 22729.56,E2 22729.56} C_VEL
LIN {X 0,Y 472.944,Z 406.808,A -85,B 0,C 180,E1 22725.928,E2 22725.928} C_VEL
LIN {X 0,Y 472.947,Z 406.811,A -85,B 0,C 180,E1 22722.244,E2 22722.244} C_VEL
LIN {X 0,Y 472.939,Z 406.82,A -85,B 0,C 180,E1 22718.727,E2 22718.727} C_VEL
LIN {X 0,Y 472.945,Z 406.819,A -85,B 0,C 180,E1 22715.097,E2 22715.097} C_VEL
LIN {X 0,Y 472.942,Z 406.809,A -85,B 0,C 180,E1 22711.48,E2 22711.48} C_VEL
LIN {X 0,Y 472.953,Z 406.817,A -85,B 0,C 180,E1 22707.854,E2 22707.854} C_VEL
LIN {X 0,Y 472.94,Z 406.819,A -85,B 0,C 180,E1 22704.214,E2 22704.214} C_VEL
LIN {X 0,Y 472.945,Z 406.806,A -85,B 0,C 180,E1 22700.517,E2 22700.517} C_VEL
LIN {X 0,Y 472.945,Z 406.824,A -85,B 0,C 180,E1 22696.836,E2 22696.836} C_VEL
LIN {X 0,Y 472.944,Z 406.812,A -85,B 0,C 180,E1 22693.199,E2 22693.199} C_VEL
LIN {X 0,Y 472.943,Z 406.808,A -85,B 0,C 180,E1 22689.615,E2 22689.615} C_VEL
LIN {X 0,Y 472.947,Z 406.823,A -85,B 0,C 180,E1 22685.946,E2 22685.946} C_VEL
LIN {X 0,Y 472.941,Z 406.808,A -85,B 0,C 180,E1 22682.302,E2 22682.302} C_VEL
LIN {X 0,Y 472.942,Z 406.813,A -85,B 0,C 180,E1 22678.668,E2 22678.668} C_VEL
LIN {X 0,Y 472.946,Z 406.819,A -85,B 0,C 180,E1 22675.028,E2 22675.028} C_VEL
LIN {X 0,Y 472.946,Z 406.819,A -85,B 0,C 180,E1 22671.368,E2 22671.368} C_VEL
LIN {X 0,Y 472.944,Z 406.81,A -85,B 0,C 180,E1 22667.671,E2 22667.671} C_VEL
LIN {X 0,Y 472.937,Z 406.818,A -85,B 0,C 180,E1 22664.048,E2 22664.048} C_VEL
LIN {X 0,Y 472.951,Z 406.818,A -85,B 0,C 180,E1 22660.359,E2 22660.359} C_VEL
LIN {X 0,Y 472.948,Z 406.821,A -85,B 0,C 180,E1 22656.713,E2 22656.713} C_VEL
LIN {X 0,Y 472.947,Z 406.826,A -85,B 0,C 180,E1 22653.101,E2 22653.101} C_VEL
LIN {X 0,Y 472.937,Z 406.825,A -85,B 0,C 180,E1 22649.51,E2 22649.51} C_VEL
LIN {X 0,Y 472.948,Z 406.82,A -85,B 0,C 180,E1 22645.928,E2 22645.928} C_VEL
LIN {X 0,Y 472.947,Z 406.814,A -85,B 0,C 180,E1 22642.25,E2 22642.25} C_VEL
LIN {X 0,Y 472.945,Z 406.821,A -85,B 0,C 180,E1 22638.636,E2 22638.636} C_VEL
LIN {X 0,Y 472.968,Z 407.065,A -85,B 0,C 180,E1 22637.124,E2 22637.124} C_VEL
LIN {X 0,Y 474.36,Z 410.464,A -85,B 0,C 180,E1 22636.596,E2 22636.596} C_VEL
LIN {X 0,Y 481.357,Z 424.93,A -85,B 0,C 180,E1 22634.564,E2 22634.564} C_VEL
LIN {X 0,Y 489.33,Z 442.573,A -85,B 0,C 180,E1 22632.296,E2 22632.296} C_VEL
LIN {X 0,Y 492.858,Z 450.982,A -85,B 0,C 180,E1 22631.294,E2 22631.294} C_VEL
LIN {X 0,Y 492.736,Z 455.809,A -85,B 0,C 180,E1 22630.987,E2 22630.987} C_VEL
LIN {X 0,Y 496.339,Z 480.456,A -85,B 0,C 180,E1 22630.21,E2 22630.21} C_VEL
LIN {X 0,Y 492.494,Z 700.009,A -85,B 0,C 180,E1 22626.667,E2 22626.667} C_VEL
LIN {X 0,Y 491.331,Z 761.685,A -85,B 0,C 180,E1 22625.657,E2 22625.657} C_VEL
LIN {X 0,Y 490.337,Z 782.783,A -85,B 0,C 180,E1 22625.114,E2 22625.114} C_VEL
LIN {X 0,Y 488.976,Z 805.082,A -85,B 0,C 180,E1 22624.323,E2 22624.323} C_VEL
LIN {X 0,Y 487.516,Z 825.565,A -85,B 0,C 180,E1 22623.386,E2 22623.386} C_VEL
LIN {X 0,Y 485.756,Z 846,A -85,B 0,C 180,E1 22622.218,E2 22622.218} C_VEL
LIN {X 0,Y 483.898,Z 866.071,A -85,B 0,C 180,E1 22620.828,E2 22620.828} C_VEL
LIN {X 0,Y 482.015,Z 885.164,A -85,B 0,C 180,E1 22619.262,E2 22619.262} C_VEL
LIN {X 0,Y 480.42,Z 900.459,A -85,B 0,C 180,E1 22617.789,E2 22617.789} C_VEL
LIN {X 0,Y 478.524,Z 917.638,A -85,B 0,C 180,E1 22615.829,E2 22615.829} C_VEL
LIN {X 0,Y 476.853,Z 933.315,A -85,B 0,C 180,E1 22613.742,E2 22613.742} C_VEL
LIN {X 0,Y 475.441,Z 947.077,A -85,B 0,C 180,E1 22611.596,E2 22611.596} C_VEL
LIN {X 0,Y 474.275,Z 959.534,A -85,B 0,C 180,E1 22609.331,E2 22609.331} C_VEL
LIN {X 0,Y 473.353,Z 970.98,A -85,B 0,C 180,E1 22606.891,E2 22606.891} C_VEL
LIN {X 0,Y 472.715,Z 980.503,A -85,B 0,C 180,E1 22604.455,E2 22604.455} C_VEL
LIN {X 0,Y 472.3,Z 988.462,A -85,B 0,C 180,E1 22601.976,E2 22601.976} C_VEL
LIN {X 0,Y 472.07,Z 994.867,A -85,B 0,C 180,E1 22599.512,E2 22599.512} C_VEL
LIN {X 0,Y 471.957,Z 999.808,A -85,B 0,C 180,E1 22596.938,E2 22596.938} C_VEL
LIN {X 0,Y 471.919,Z 1003.33,A -85,B 0,C 180,E1 22594.255,E2 22594.255} C_VEL
LIN {X 0,Y 471.9,Z 1005.15,A -85,B 0,C 180,E1 22591.702,E2 22591.702} C_VEL
LIN {X 0,Y 471.897,Z 1005.349,A -85,B 0,C 180,E1 22589.153,E2 22589.153} C_VEL
LIN {X 0,Y 471.912,Z 1004.125,A -85,B 0,C 180,E1 22586.602,E2 22586.602} C_VEL
LIN {X 0,Y 471.941,Z 1001.301,A -85,B 0,C 180,E1 22584.044,E2 22584.044} C_VEL
LIN {X 0,Y 472.026,Z 996.658,A -85,B 0,C 180,E1 22581.353,E2 22581.353} C_VEL
LIN {X 0,Y 472.224,Z 990.596,A -85,B 0,C 180,E1 22578.77,E2 22578.77} C_VEL
LIN {X 0,Y 472.578,Z 983.08,A -85,B 0,C 180,E1 22576.296,E2 22576.296} C_VEL
LIN {X 0,Y 473.187,Z 973.335,A -85,B 0,C 180,E1 22573.681,E2 22573.681} C_VEL
LIN {X 0,Y 474.03,Z 962.583,A -85,B 0,C 180,E1 22571.273,E2 22571.273} C_VEL
LIN {X 0,Y 475.156,Z 950.074,A -85,B 0,C 180,E1 22568.914,E2 22568.914} C_VEL
LIN {X 0,Y 476.47,Z 936.731,A -85,B 0,C 180,E1 22566.768,E2 22566.768} C_VEL
LIN {X 0,Y 478.086,Z 921.735,A -85,B 0,C 180,E1 22564.683,E2 22564.683} C_VEL
LIN {X 0,Y 479.918,Z 905.27,A -85,B 0,C 180,E1 22562.723,E2 22562.723} C_VEL
LIN {X 0,Y 481.549,Z 889.574,A -85,B 0,C 180,E1 22561.146,E2 22561.146} C_VEL
LIN {X 0,Y 483.415,Z 871.02,A -85,B 0,C 180,E1 22559.557,E2 22559.557} C_VEL
LIN {X 0,Y 485.185,Z 851.681,A -85,B 0,C 180,E1 22558.163,E2 22558.163} C_VEL
LIN {X 0,Y 486.912,Z 831.732,A -85,B 0,C 180,E1 22556.966,E2 22556.966} C_VEL
LIN {X 0,Y 488.473,Z 811.54,A -85,B 0,C 180,E1 22555.967,E2 22555.967} C_VEL
LIN {X 0,Y 489.81,Z 789.853,A -85,B 0,C 180,E1 22555.132,E2 22555.132} C_VEL
LIN {X 0,Y 490.914,Z 768.077,A -85,B 0,C 180,E1 22554.516,E2 22554.516} C_VEL
LIN {X 0,Y 491.636,Z 744.648,A -85,B 0,C 180,E1 22554.067,E2 22554.067} C_VEL
LIN {X 0,Y 495.452,Z 512.642,A -85,B 0,C 180,E1 22550.365,E2 22550.365} C_VEL
LIN {X 0,Y 495.85,Z 478.01,A -85,B 0,C 180,E1 22549.783,E2 22549.783} C_VEL
LIN {X 0,Y 492.318,Z 454.392,A -85,B 0,C 180,E1 22549.01,E2 22549.01} C_VEL
LIN {X 0,Y 492.469,Z 450.133,A -85,B 0,C 180,E1 22548.695,E2 22548.695} C_VEL
LIN {X 0,Y 482.123,Z 426.534,A -85,B 0,C 180,E1 22545.767,E2 22545.767} C_VEL
LIN {X 0,Y 474.594,Z 410.818,A -85,B 0,C 180,E1 22543.544,E2 22543.544} C_VEL
LIN {X 0,Y 472.994,Z 407.29,A -85,B 0,C 180,E1 22543.001,E2 22543.001} C_VEL
LIN {X 0,Y 472.946,Z 406.805,A -85,B 0,C 180,E1 22542.407,E2 22542.407} C_VEL
LIN {X 0,Y 472.913,Z 406.826,A -85,B 0,C 180,E1 22538.897,E2 22538.897} C_VEL
LIN {X 0,Y 472.912,Z 406.828,A -85,B 0,C 180,E1 22535.253,E2 22535.253} C_VEL
LIN {X 0,Y 472.951,Z 406.819,A -85,B 0,C 180,E1 22531.763,E2 22531.763} C_VEL
LIN {X 0,Y 472.916,Z 406.825,A -85,B 0,C 180,E1 22528.267,E2 22528.267} C_VEL
LIN {X 0,Y 472.888,Z 406.828,A -85,B 0,C 180,E1 22524.749,E2 22524.749} C_VEL
LIN {X 0,Y 472.905,Z 406.821,A -85,B 0,C 180,E1 22521.199,E2 22521.199} C_VEL
LIN {X 0,Y 472.924,Z 406.82,A -85,B 0,C 180,E1 22517.724,E2 22517.724} C_VEL
LIN {X 0,Y 472.87,Z 406.824,A -85,B 0,C 180,E1 22514.323,E2 22514.323} C_VEL
LIN {X 0,Y 472.883,Z 406.829,A -85,B 0,C 180,E1 22510.723,E2 22510.723} C_VEL
LIN {X 0,Y 472.936,Z 406.825,A -85,B 0,C 180,E1 22507.165,E2 22507.165} C_VEL
LIN {X 0,Y 472.915,Z 406.828,A -85,B 0,C 180,E1 22503.636,E2 22503.636} C_VEL
LIN {X 0,Y 472.896,Z 406.828,A -85,B 0,C 180,E1 22500.121,E2 22500.121} C_VEL
LIN {X 0,Y 472.923,Z 406.818,A -85,B 0,C 180,E1 22496.606,E2 22496.606} C_VEL
LIN {X 0,Y 472.955,Z 406.819,A -85,B 0,C 180,E1 22493.079,E2 22493.079} C_VEL
LIN {X 0,Y 472.929,Z 406.827,A -85,B 0,C 180,E1 22489.426,E2 22489.426} C_VEL
LIN {X 0,Y 472.916,Z 406.825,A -85,B 0,C 180,E1 22485.803,E2 22485.803} C_VEL
LIN {X 0,Y 472.943,Z 406.82,A -85,B 0,C 180,E1 22482.276,E2 22482.276} C_VEL
LIN {X 0,Y 472.975,Z 407.09,A -85,B 0,C 180,E1 22479.285,E2 22479.285} C_VEL
LIN {X 0,Y 474.612,Z 410.826,A -85,B 0,C 180,E1 22478.625,E2 22478.625} C_VEL
LIN {X 0,Y 482.617,Z 429.123,A -85,B 0,C 180,E1 22475.782,E2 22475.782} C_VEL
LIN {X 0,Y 489.116,Z 445.961,A -85,B 0,C 180,E1 22473.437,E2 22473.437} C_VEL
LIN {X 0,Y 488.686,Z 453.222,A -85,B 0,C 180,E1 22472.821,E2 22472.821} C_VEL
LIN {X 0,Y 492.937,Z 476.821,A -85,B 0,C 180,E1 22471.971,E2 22471.971} C_VEL
LIN {X 0,Y 487.884,Z 717.529,A -85,B 0,C 180,E1 22467.978,E2 22467.978} C_VEL
LIN {X 0,Y 487.697,Z 721.698,A -85,B 0,C 180,E1 22467.879,E2 22467.879} C_VEL
LIN {X 0,Y 486.211,Z 730.382,A -85,B 0,C 180,E1 22467.744,E2 22467.744} C_VEL
LIN {X 0,Y 480.761,Z 747.333,A -85,B 0,C 180,E1 22467.544,E2 22467.544} C_VEL
LIN {X 0,Y 479.285,Z 754.733,A -85,B 0,C 180,E1 22467.325,E2 22467.325} C_VEL
LIN {X 0,Y 479.199,Z 755.746,A -85,B 0,C 180,E1 22467.282,E2 22467.282} C_VEL
LIN {X 0,Y 477.838,Z 774.471,A -85,B 0,C 180,E1 22466.38,E2 22466.38} C_VEL
LIN {X 0,Y 476.196,Z 793.361,A -85,B 0,C 180,E1 22465.238,E2 22465.238} C_VEL
LIN {X 0,Y 474.425,Z 811.233,A -85,B 0,C 180,E1 22463.902,E2 22463.902} C_VEL
LIN {X 0,Y 472.609,Z 828.186,A -85,B 0,C 180,E1 22462.38,E2 22462.38} C_VEL
LIN {X 0,Y 470.778,Z 844.56,A -85,B 0,C 180,E1 22460.625,E2 22460.625} C_VEL
LIN {X 0,Y 469.094,Z 859.682,A -85,B 0,C 180,E1 22458.692,E2 22458.692} C_VEL
LIN {X 0,Y 467.632,Z 873.094,A -85,B 0,C 180,E1 22456.658,E2 22456.658} C_VEL
LIN {X 0,Y 466.394,Z 885.342,A -85,B 0,C 180,E1 22454.447,E2 22454.447} C_VEL
LIN {X 0,Y 465.413,Z 896.201,A -85,B 0,C 180,E1 22452.083,E2 22452.083} C_VEL
LIN {X 0,Y 464.714,Z 905.377,A -85,B 0,C 180,E1 22449.622,E2 22449.622} C_VEL
LIN {X 0,Y 464.282,Z 912.65,A -85,B 0,C 180,E1 22447.172,E2 22447.172} C_VEL
LIN {X 0,Y 464.052,Z 918.352,A -85,B 0,C 180,E1 22444.664,E2 22444.664} C_VEL
LIN {X 0,Y 463.944,Z 922.452,A -85,B 0,C 180,E1 22442.116,E2 22442.116} C_VEL
LIN {X 0,Y 463.923,Z 924.849,A -85,B 0,C 180,E1 22439.708,E2 22439.708} C_VEL
LIN {X 0,Y 463.911,Z 925.765,A -85,B 0,C 180,E1 22437.109,E2 22437.109} C_VEL
LIN {X 0,Y 463.919,Z 925.031,A -85,B 0,C 180,E1 22434.561,E2 22434.561} C_VEL
LIN {X 0,Y 463.947,Z 922.71,A -85,B 0,C 180,E1 22432.02,E2 22432.02} C_VEL
LIN {X 0,Y 464.028,Z 918.822,A -85,B 0,C 180,E1 22429.507,E2 22429.507} C_VEL
LIN {X 0,Y 464.245,Z 913.314,A -85,B 0,C 180,E1 22427.008,E2 22427.008} C_VEL
LIN {X 0,Y 464.659,Z 905.836,A -85,B 0,C 180,E1 22424.451,E2 22424.451} C_VEL
LIN {X 0,Y 465.311,Z 896.833,A -85,B 0,C 180,E1 22422.027,E2 22422.027} C_VEL
LIN {X 0,Y 466.202,Z 886.512,A -85,B 0,C 180,E1 22419.752,E2 22419.752} C_VEL
LIN {X 0,Y 467.335,Z 874.953,A -85,B 0,C 180,E1 22417.62,E2 22417.62} C_VEL
LIN {X 0,Y 468.781,Z 861.313,A -85,B 0,C 180,E1 22415.505,E2 22415.505} C_VEL
LIN {X 0,Y 470.345,Z 847.195,A -85,B 0,C 180,E1 22413.654,E2 22413.654} C_VEL
LIN {X 0,Y 472.121,Z 831.136,A -85,B 0,C 180,E1 22411.878,E2 22411.878} C_VEL
LIN {X 0,Y 473.988,Z 813.314,A -85,B 0,C 180,E1 22410.239,E2 22410.239} C_VEL
LIN {X 0,Y 475.737,Z 795.307,A -85,B 0,C 180,E1 22408.872,E2 22408.872} C_VEL
LIN {X 0,Y 477.356,Z 776.699,A -85,B 0,C 180,E1 22407.717,E2 22407.717} C_VEL
LIN {X 0,Y 478.835,Z 756.846,A -85,B 0,C 180,E1 22406.736,E2 22406.736} C_VEL
LIN {X 0,Y 480.029,Z 736.943,A -85,B 0,C 180,E1 22405.985,E2 22405.985} C_VEL
LIN {X 0,Y 480.946,Z 716.431,A -85,B 0,C 180,E1 22405.437,E2 22405.437} C_VEL
LIN {X 0,Y 485.908,Z 477.505,A -85,B 0,C 180,E1 22401.478,E2 22401.478} C_VEL
LIN {X 0,Y 481.354,Z 452.259,A -85,B 0,C 180,E1 22400.553,E2 22400.553} C_VEL
LIN {X 0,Y 481.574,Z 448.259,A -85,B 0,C 180,E1 22400.195,E2 22400.195} C_VEL
LIN {X 0,Y 474.114,Z 429.226,A -85,B 0,C 180,E1 22397.535,E2 22397.535} C_VEL
LIN {X 0,Y 467.818,Z 414.724,A -85,B 0,C 180,E1 22395.327,E2 22395.327} C_VEL
LIN {X 0,Y 465.021,Z 407.994,A -85,B 0,C 180,E1 22394.223,E2 22394.223} C_VEL
LIN {X 0,Y 465.01,Z 407.802,A -85,B 0,C 180,E1 22390.724,E2 22390.724} C_VEL
LIN {X 0,Y 465.007,Z 407.765,A -85,B 0,C 180,E1 22386.96,E2 22386.96} C_VEL
LIN {X 0,Y 465.005,Z 407.809,A -85,B 0,C 180,E1 22383.293,E2 22383.293} C_VEL
LIN {X 0,Y 464.997,Z 407.803,A -85,B 0,C 180,E1 22379.571,E2 22379.571} C_VEL
LIN {X 0,Y 465.005,Z 407.802,A -85,B 0,C 180,E1 22375.859,E2 22375.859} C_VEL
LIN {X 0,Y 465.007,Z 407.809,A -85,B 0,C 180,E1 22372.205,E2 22372.205} C_VEL
LIN {X 0,Y 465.014,Z 407.808,A -85,B 0,C 180,E1 22368.526,E2 22368.526} C_VEL
LIN {X 0,Y 465.004,Z 407.809,A -85,B 0,C 180,E1 22364.798,E2 22364.798} C_VEL
LIN {X 0,Y 465.003,Z 407.8,A -85,B 0,C 180,E1 22361.146,E2 22361.146} C_VEL
LIN {X 0,Y 465.008,Z 407.8,A -85,B 0,C 180,E1 22357.482,E2 22357.482} C_VEL
LIN {X 0,Y 465.007,Z 407.81,A -85,B 0,C 180,E1 22353.842,E2 22353.842} C_VEL
LIN {X 0,Y 465.01,Z 407.802,A -85,B 0,C 180,E1 22350.186,E2 22350.186} C_VEL
LIN {X 0,Y 465.002,Z 407.795,A -85,B 0,C 180,E1 22346.554,E2 22346.554} C_VEL
LIN {X 0,Y 465.011,Z 407.812,A -85,B 0,C 180,E1 22342.904,E2 22342.904} C_VEL
LIN {X 0,Y 465.002,Z 407.797,A -85,B 0,C 180,E1 22339.208,E2 22339.208} C_VEL
LIN {X 0,Y 465.013,Z 407.8,A -85,B 0,C 180,E1 22335.572,E2 22335.572} C_VEL
LIN {X 0,Y 465.003,Z 407.812,A -85,B 0,C 180,E1 22331.913,E2 22331.913} C_VEL
LIN {X 0,Y 465.009,Z 407.796,A -85,B 0,C 180,E1 22328.159,E2 22328.159} C_VEL
LIN {X 0,Y 465,Z 407.807,A -85,B 0,C 180,E1 22324.564,E2 22324.564} C_VEL
LIN {X 0,Y 465.009,Z 407.807,A -85,B 0,C 180,E1 22320.863,E2 22320.863} C_VEL
LIN {X 0,Y 465.006,Z 407.8,A -85,B 0,C 180,E1 22317.166,E2 22317.166} C_VEL
LIN {X 0,Y 465.005,Z 407.796,A -85,B 0,C 180,E1 22313.419,E2 22313.419} C_VEL
LIN {X 0,Y 465.007,Z 407.813,A -85,B 0,C 180,E1 22309.72,E2 22309.72} C_VEL
LIN {X 0,Y 464.998,Z 407.809,A -85,B 0,C 180,E1 22306.065,E2 22306.065} C_VEL
LIN {X 0,Y 465.01,Z 407.804,A -85,B 0,C 180,E1 22302.481,E2 22302.481} C_VEL
LIN {X 0,Y 465.007,Z 407.8,A -85,B 0,C 180,E1 22298.824,E2 22298.824} C_VEL
LIN {X 0,Y 465.007,Z 407.801,A -85,B 0,C 180,E1 22295.149,E2 22295.149} C_VEL
LIN {X 0,Y 464.997,Z 407.802,A -85,B 0,C 180,E1 22291.488,E2 22291.488} C_VEL
LIN {X 0,Y 465.01,Z 407.8,A -85,B 0,C 180,E1 22287.908,E2 22287.908} C_VEL
LIN {X 0,Y 465.01,Z 407.808,A -85,B 0,C 180,E1 22284.159,E2 22284.159} C_VEL
LIN {X 0,Y 465.018,Z 407.809,A -85,B 0,C 180,E1 22280.473,E2 22280.473} C_VEL
LIN {X 0,Y 465.052,Z 408.108,A -85,B 0,C 180,E1 22277.97,E2 22277.97} C_VEL
LIN {X 0,Y 466.694,Z 411.836,A -85,B 0,C 180,E1 22277.39,E2 22277.39} C_VEL
LIN {X 0,Y 475.008,Z 429.047,A -85,B 0,C 180,E1 22274.903,E2 22274.903} C_VEL
LIN {X 0,Y 483.315,Z 447.633,A -85,B 0,C 180,E1 22272.481,E2 22272.481} C_VEL
LIN {X 0,Y 486.136,Z 454.377,A -85,B 0,C 180,E1 22271.664,E2 22271.664} C_VEL
LIN {X 0,Y 490,Z 481.766,A -85,B 0,C 180,E1 22270.763,E2 22270.763} C_VEL
LIN {X 0,Y 485.862,Z 701.002,A -85,B 0,C 180,E1 22267.181,E2 22267.181} C_VEL
LIN {X 0,Y 484.64,Z 761.269,A -85,B 0,C 180,E1 22266.182,E2 22266.182} C_VEL
LIN {X 0,Y 483.58,Z 782.471,A -85,B 0,C 180,E1 22265.631,E2 22265.631} C_VEL
LIN {X 0,Y 482.163,Z 804.382,A -85,B 0,C 180,E1 22264.847,E2 22264.847} C_VEL
LIN {X 0,Y 480.557,Z 825.235,A -85,B 0,C 180,E1 22263.884,E2 22263.884} C_VEL
LIN {X 0,Y 478.702,Z 845.59,A -85,B 0,C 180,E1 22262.706,E2 22262.706} C_VEL
LIN {X 0,Y 476.757,Z 865.095,A -85,B 0,C 180,E1 22261.341,E2 22261.341} C_VEL
LIN {X 0,Y 474.815,Z 883.746,A -85,B 0,C 180,E1 22259.801,E2 22259.801} C_VEL
LIN {X 0,Y 472.842,Z 901.553,A -85,B 0,C 180,E1 22258.068,E2 22258.068} C_VEL
LIN {X 0,Y 471.033,Z 917.994,A -85,B 0,C 180,E1 22256.203,E2 22256.203} C_VEL
LIN {X 0,Y 469.598,Z 930.63,A -85,B 0,C 180,E1 22254.533,E2 22254.533} C_VEL
LIN {X 0,Y 467.988,Z 944.984,A -85,B 0,C 180,E1 22252.317,E2 22252.317} C_VEL
LIN {X 0,Y 466.637,Z 958.263,A -85,B 0,C 180,E1 22249.921,E2 22249.921} C_VEL
LIN {X 0,Y 465.625,Z 969.666,A -85,B 0,C 180,E1 22247.498,E2 22247.498} C_VEL
LIN {X 0,Y 464.869,Z 979.584,A -85,B 0,C 180,E1 22244.96,E2 22244.96} C_VEL
LIN {X 0,Y 464.361,Z 988.108,A -85,B 0,C 180,E1 22242.31,E2 22242.31} C_VEL
LIN {X 0,Y 464.091,Z 994.577,A -85,B 0,C 180,E1 22239.802,E2 22239.802} C_VEL
LIN {X 0,Y 463.956,Z 999.395,A -85,B 0,C 180,E1 22237.307,E2 22237.307} C_VEL
LIN {X 0,Y 463.91,Z 1002.874,A -85,B 0,C 180,E1 22234.824,E2 22234.824} C_VEL
LIN {X 0,Y 463.908,Z 1004.881,A -85,B 0,C 180,E1 22232.226,E2 22232.226} C_VEL
LIN {X 0,Y 463.894,Z 1005.417,A -85,B 0,C 180,E1 22229.509,E2 22229.509} C_VEL
LIN {X 0,Y 463.898,Z 1004.473,A -85,B 0,C 180,E1 22227.038,E2 22227.038} C_VEL
LIN {X 0,Y 463.925,Z 1001.94,A -85,B 0,C 180,E1 22224.437,E2 22224.437} C_VEL
LIN {X 0,Y 464.015,Z 997.928,A -85,B 0,C 180,E1 22221.827,E2 22221.827} C_VEL
LIN {X 0,Y 464.195,Z 992.166,A -85,B 0,C 180,E1 22219.202,E2 22219.202} C_VEL
LIN {X 0,Y 464.553,Z 984.7,A -85,B 0,C 180,E1 22216.562,E2 22216.562} C_VEL
LIN {X 0,Y 465.14,Z 975.906,A -85,B 0,C 180,E1 22214.032,E2 22214.032} C_VEL
LIN {X 0,Y 466.009,Z 965.106,A -85,B 0,C 180,E1 22211.489,E2 22211.489} C_VEL
LIN {X 0,Y 467.168,Z 952.875,A -85,B 0,C 180,E1 22209.061,E2 22209.061} C_VEL
LIN {X 0,Y 468.621,Z 939.265,A -85,B 0,C 180,E1 22206.755,E2 22206.755} C_VEL
LIN {X 0,Y 470.361,Z 924.189,A -85,B 0,C 180,E1 22204.574,E2 22204.574} C_VEL
LIN {X 0,Y 472.044,Z 908.621,A -85,B 0,C 180,E1 22202.708,E2 22202.708} C_VEL
LIN {X 0,Y 474.017,Z 890.48,A -85,B 0,C 180,E1 22200.839,E2 22200.839} C_VEL
LIN {X 0,Y 476.062,Z 871.525,A -85,B 0,C 180,E1 22199.176,E2 22199.176} C_VEL
LIN {X 0,Y 477.934,Z 852.327,A -85,B 0,C 180,E1 22197.764,E2 22197.764} C_VEL
LIN {X 0,Y 479.876,Z 831.52,A -85,B 0,C 180,E1 22196.49,E2 22196.49} C_VEL
LIN {X 0,Y 481.542,Z 811.278,A -85,B 0,C 180,E1 22195.474,E2 22195.474} C_VEL
LIN {X 0,Y 482.976,Z 789.587,A -85,B 0,C 180,E1 22194.628,E2 22194.628} C_VEL
LIN {X 0,Y 484.161,Z 767.775,A -85,B 0,C 180,E1 22194.004,E2 22194.004} C_VEL
LIN {X 0,Y 484.923,Z 744.465,A -85,B 0,C 180,E1 22193.551,E2 22193.551} C_VEL
LIN {X 0,Y 489.014,Z 513.769,A -85,B 0,C 180,E1 22189.823,E2 22189.823} C_VEL
LIN {X 0,Y 489.482,Z 479.509,A -85,B 0,C 180,E1 22189.24,E2 22189.24} C_VEL
LIN {X 0,Y 485.789,Z 454.459,A -85,B 0,C 180,E1 22188.409,E2 22188.409} C_VEL
LIN {X 0,Y 484.721,Z 451.423,A -85,B 0,C 180,E1 22188.067,E2 22188.067} C_VEL
LIN {X 0,Y 476.164,Z 431.599,A -85,B 0,C 180,E1 22185.556,E2 22185.556} C_VEL
LIN {X 0,Y 468.922,Z 416.264,A -85,B 0,C 180,E1 22183.36,E2 22183.36} C_VEL
LIN {X 0,Y 465.103,Z 408.351,A -85,B 0,C 180,E1 22182.111,E2 22182.111} C_VEL
LIN {X 0,Y 464.996,Z 407.806,A -85,B 0,C 180,E1 22181.638,E2 22181.638} C_VEL
LIN {X 0,Y 465.019,Z 407.808,A -85,B 0,C 180,E1 22178.104,E2 22178.104} C_VEL
LIN {X 0,Y 464.984,Z 407.811,A -85,B 0,C 180,E1 22174.439,E2 22174.439} C_VEL
LIN {X 0,Y 464.961,Z 407.818,A -85,B 0,C 180,E1 22170.914,E2 22170.914} C_VEL
LIN {X 0,Y 464.979,Z 407.811,A -85,B 0,C 180,E1 22167.375,E2 22167.375} C_VEL
LIN {X 0,Y 465,Z 407.807,A -85,B 0,C 180,E1 22163.843,E2 22163.843} C_VEL
LIN {X 0,Y 464.947,Z 407.813,A -85,B 0,C 180,E1 22160.359,E2 22160.359} C_VEL
LIN {X 0,Y 464.938,Z 407.819,A -85,B 0,C 180,E1 22156.748,E2 22156.748} C_VEL
LIN {X 0,Y 464.984,Z 407.818,A -85,B 0,C 180,E1 22153.302,E2 22153.302} C_VEL
LIN {X 0,Y 464.976,Z 407.818,A -85,B 0,C 180,E1 22149.655,E2 22149.655} C_VEL
LIN {X 0,Y 464.947,Z 407.818,A -85,B 0,C 180,E1 22146.172,E2 22146.172} C_VEL
LIN {X 0,Y 464.956,Z 407.811,A -85,B 0,C 180,E1 22142.465,E2 22142.465} C_VEL
LIN {X 0,Y 465.011,Z 407.806,A -85,B 0,C 180,E1 22139.014,E2 22139.014} C_VEL
LIN {X 0,Y 464.998,Z 407.811,A -85,B 0,C 180,E1 22135.313,E2 22135.313} C_VEL
LIN {X 0,Y 464.973,Z 407.816,A -85,B 0,C 180,E1 22131.716,E2 22131.716} C_VEL
LIN {X 0,Y 464.979,Z 407.813,A -85,B 0,C 180,E1 22128.049,E2 22128.049} C_VEL
LIN {X 0,Y 465.008,Z 407.808,A -85,B 0,C 180,E1 22124.408,E2 22124.408} C_VEL
LIN {X 0,Y 465.015,Z 407.808,A -85,B 0,C 180,E1 22120.708,E2 22120.708} C_VEL
LIN {X 0,Y 465.067,Z 408.243,A -85,B 0,C 180,E1 22120.158,E2 22120.158} C_VEL
LIN {X 0,Y 466.519,Z 411.632,A -85,B 0,C 180,E1 22119.552,E2 22119.552} C_VEL
LIN {X 0,Y 473.6,Z 427.264,A -85,B 0,C 180,E1 22116.985,E2 22116.985} C_VEL
LIN {X 0,Y 481.089,Z 445.841,A -85,B 0,C 180,E1 22114.254,E2 22114.254} C_VEL
LIN {X 0,Y 482.332,Z 449.158,A -85,B 0,C 180,E1 22113.797,E2 22113.797} C_VEL
LIN {X 0,Y 482.187,Z 453.475,A -85,B 0,C 180,E1 22113.449,E2 22113.449} C_VEL
LIN {X 0,Y 486.639,Z 478.354,A -85,B 0,C 180,E1 22112.531,E2 22112.531} C_VEL
LIN {X 0,Y 481.199,Z 718.044,A -85,B 0,C 180,E1 22108.494,E2 22108.494} C_VEL
LIN {X 0,Y 480.225,Z 739.033,A -85,B 0,C 180,E1 22107.917,E2 22107.917} C_VEL
LIN {X 0,Y 479.199,Z 755.746,A -85,B 0,C 180,E1 22107.282,E2 22107.282} C_VEL
LIN {X 0,Y 477.875,Z 763.183,A -85,B 0,C 180,E1 22107.018,E2 22107.018} C_VEL
LIN {X 0,Y 471.27,Z 781.539,A -85,B 0,C 180,E1 22106.445,E2 22106.445} C_VEL
LIN {X 0,Y 469.765,Z 788.444,A -85,B 0,C 180,E1 22106.082,E2 22106.082} C_VEL
LIN {X 0,Y 467.987,Z 805.972,A -85,B 0,C 180,E1 22104.845,E2 22104.845} C_VEL
LIN {X 0,Y 466.071,Z 823.501,A -85,B 0,C 180,E1 22103.347,E2 22103.347} C_VEL
LIN {X 0,Y 464.106,Z 840.104,A -85,B 0,C 180,E1 22101.64,E2 22101.64} C_VEL
LIN {X 0,Y 462.248,Z 855.341,A -85,B 0,C 180,E1 22099.772,E2 22099.772} C_VEL
LIN {X 0,Y 460.584,Z 869.263,A -85,B 0,C 180,E1 22097.748,E2 22097.748} C_VEL
LIN {X 0,Y 459.157,Z 881.84,A -85,B 0,C 180,E1 22095.576,E2 22095.576} C_VEL
LIN {X 0,Y 458,Z 893.014,A -85,B 0,C 180,E1 22093.269,E2 22093.269} C_VEL
LIN {X 0,Y 457.192,Z 902.171,A -85,B 0,C 180,E1 22090.997,E2 22090.997} C_VEL
LIN {X 0,Y 456.55,Z 910.685,A -85,B 0,C 180,E1 22088.368,E2 22088.368} C_VEL
LIN {X 0,Y 456.209,Z 917.062,A -85,B 0,C 180,E1 22085.811,E2 22085.811} C_VEL
LIN {X 0,Y 456.038,Z 921.765,A -85,B 0,C 180,E1 22083.234,E2 22083.234} C_VEL
LIN {X 0,Y 455.959,Z 924.902,A -85,B 0,C 180,E1 22080.576,E2 22080.576} C_VEL
LIN {X 0,Y 455.947,Z 926.336,A -85,B 0,C 180,E1 22077.984,E2 22077.984} C_VEL
LIN {X 0,Y 455.944,Z 926.189,A -85,B 0,C 180,E1 22075.378,E2 22075.378} C_VEL
LIN {X 0,Y 455.974,Z 924.441,A -85,B 0,C 180,E1 22072.834,E2 22072.834} C_VEL
LIN {X 0,Y 456.05,Z 921.062,A -85,B 0,C 180,E1 22070.264,E2 22070.264} C_VEL
LIN {X 0,Y 456.228,Z 916.125,A -85,B 0,C 180,E1 22067.732,E2 22067.732} C_VEL
LIN {X 0,Y 456.588,Z 909.597,A -85,B 0,C 180,E1 22065.232,E2 22065.232} C_VEL
LIN {X 0,Y 457.205,Z 901.326,A -85,B 0,C 180,E1 22062.745,E2 22062.745} C_VEL
LIN {X 0,Y 458.11,Z 891.279,A -85,B 0,C 180,E1 22060.307,E2 22060.307} C_VEL
LIN {X 0,Y 459.337,Z 879.358,A -85,B 0,C 180,E1 22057.935,E2 22057.935} C_VEL
LIN {X 0,Y 460.73,Z 866.809,A -85,B 0,C 180,E1 22055.851,E2 22055.851} C_VEL
LIN {X 0,Y 462.402,Z 852.483,A -85,B 0,C 180,E1 22053.841,E2 22053.841} C_VEL
LIN {X 0,Y 464.261,Z 836.659,A -85,B 0,C 180,E1 22051.972,E2 22051.972} C_VEL
LIN {X 0,Y 466.132,Z 820.487,A -85,B 0,C 180,E1 22050.366,E2 22050.366} C_VEL
LIN {X 0,Y 468.034,Z 802.803,A -85,B 0,C 180,E1 22048.896,E2 22048.896} C_VEL
LIN {X 0,Y 469.876,Z 784.013,A -85,B 0,C 180,E1 22047.619,E2 22047.619} C_VEL
LIN {X 0,Y 471.437,Z 765.201,A -85,B 0,C 180,E1 22046.593,E2 22046.593} C_VEL
LIN {X 0,Y 472.82,Z 745.287,A -85,B 0,C 180,E1 22045.745,E2 22045.745} C_VEL
LIN {X 0,Y 473.915,Z 724.286,A -85,B 0,C 180,E1 22045.092,E2 22045.092} C_VEL
LIN {X 0,Y 474.649,Z 701.678,A -85,B 0,C 180,E1 22044.634,E2 22044.634} C_VEL
LIN {X 0,Y 479.51,Z 478.714,A -85,B 0,C 180,E1 22040.91,E2 22040.91} C_VEL
LIN {X 0,Y 474.773,Z 452.47,A -85,B 0,C 180,E1 22039.931,E2 22039.931} C_VEL
LIN {X 0,Y 473.829,Z 449.19,A -85,B 0,C 180,E1 22039.528,E2 22039.528} C_VEL
LIN {X 0,Y 466.282,Z 430.198,A -85,B 0,C 180,E1 22036.787,E2 22036.787} C_VEL
LIN {X 0,Y 459.761,Z 415.453,A -85,B 0,C 180,E1 22034.454,E2 22034.454} C_VEL
LIN {X 0,Y 457.114,Z 409.07,A -85,B 0,C 180,E1 22033.376,E2 22033.376} C_VEL
LIN {X 0,Y 457.068,Z 408.77,A -85,B 0,C 180,E1 22031.372,E2 22031.372} C_VEL
LIN {X 0,Y 457.051,Z 408.755,A -85,B 0,C 180,E1 22027.725,E2 22027.725} C_VEL
LIN {X 0,Y 457.066,Z 408.803,A -85,B 0,C 180,E1 22024.039,E2 22024.039} C_VEL
LIN {X 0,Y 457.075,Z 408.8,A -85,B 0,C 180,E1 22020.279,E2 22020.279} C_VEL
LIN {X 0,Y 457.071,Z 408.801,A -85,B 0,C 180,E1 22016.545,E2 22016.545} C_VEL
LIN {X 0,Y 457.071,Z 408.798,A -85,B 0,C 180,E1 22012.775,E2 22012.775} C_VEL
LIN {X 0,Y 457.059,Z 408.801,A -85,B 0,C 180,E1 22009.147,E2 22009.147} C_VEL
LIN {X 0,Y 457.064,Z 408.792,A -85,B 0,C 180,E1 22005.394,E2 22005.394} C_VEL
LIN {X 0,Y 457.068,Z 408.784,A -85,B 0,C 180,E1 22001.684,E2 22001.684} C_VEL
LIN {X 0,Y 457.068,Z 408.797,A -85,B 0,C 180,E1 21997.931,E2 21997.931} C_VEL
LIN {X 0,Y 457.07,Z 408.798,A -85,B 0,C 180,E1 21994.208,E2 21994.208} C_VEL
LIN {X 0,Y 457.063,Z 408.79,A -85,B 0,C 180,E1 21990.467,E2 21990.467} C_VEL
LIN {X 0,Y 457.07,Z 408.785,A -85,B 0,C 180,E1 21986.785,E2 21986.785} C_VEL
LIN {X 0,Y 457.068,Z 408.8,A -85,B 0,C 180,E1 21983.053,E2 21983.053} C_VEL
LIN {X 0,Y 457.064,Z 408.784,A -85,B 0,C 180,E1 21979.289,E2 21979.289} C_VEL
LIN {X 0,Y 457.073,Z 408.789,A -85,B 0,C 180,E1 21975.609,E2 21975.609} C_VEL
LIN {X 0,Y 457.064,Z 408.8,A -85,B 0,C 180,E1 21971.867,E2 21971.867} C_VEL
LIN {X 0,Y 457.07,Z 408.784,A -85,B 0,C 180,E1 21968.175,E2 21968.175} C_VEL
LIN {X 0,Y 457.062,Z 408.794,A -85,B 0,C 180,E1 21964.517,E2 21964.517} C_VEL
LIN {X 0,Y 457.065,Z 408.797,A -85,B 0,C 180,E1 21960.752,E2 21960.752} C_VEL
LIN {X 0,Y 457.067,Z 408.789,A -85,B 0,C 180,E1 21957.116,E2 21957.116} C_VEL
LIN {X 0,Y 457.066,Z 408.783,A -85,B 0,C 180,E1 21953.342,E2 21953.342} C_VEL
LIN {X 0,Y 457.069,Z 408.8,A -85,B 0,C 180,E1 21949.667,E2 21949.667} C_VEL
LIN {X 0,Y 457.06,Z 408.799,A -85,B 0,C 180,E1 21945.947,E2 21945.947} C_VEL
LIN {X 0,Y 457.07,Z 408.793,A -85,B 0,C 180,E1 21942.298,E2 21942.298} C_VEL
LIN {X 0,Y 457.07,Z 408.789,A -85,B 0,C 180,E1 21938.573,E2 21938.573} C_VEL
LIN {X 0,Y 457.071,Z 408.789,A -85,B 0,C 180,E1 21934.889,E2 21934.889} C_VEL
LIN {X 0,Y 457.061,Z 408.79,A -85,B 0,C 180,E1 21931.232,E2 21931.232} C_VEL
LIN {X 0,Y 457.061,Z 408.791,A -85,B 0,C 180,E1 21927.592,E2 21927.592} C_VEL
LIN {X 0,Y 457.071,Z 408.801,A -85,B 0,C 180,E1 21923.825,E2 21923.825} C_VEL
LIN {X 0,Y 457.071,Z 408.795,A -85,B 0,C 180,E1 21920.138,E2 21920.138} C_VEL
LIN {X 0,Y 457.094,Z 409.058,A -85,B 0,C 180,E1 21918.895,E2 21918.895} C_VEL
LIN {X 0,Y 458.607,Z 412.613,A -85,B 0,C 180,E1 21918.321,E2 21918.321} C_VEL
LIN {X 0,Y 465.792,Z 427.199,A -85,B 0,C 180,E1 21916.105,E2 21916.105} C_VEL
LIN {X 0,Y 474.384,Z 445.91,A -85,B 0,C 180,E1 21913.528,E2 21913.528} C_VEL
LIN {X 0,Y 478.513,Z 455.404,A -85,B 0,C 180,E1 21912.362,E2 21912.362} C_VEL
LIN {X 0,Y 480.213,Z 458.726,A -85,B 0,C 180,E1 21912.124,E2 21912.124} C_VEL
LIN {X 0,Y 483.697,Z 483.199,A -85,B 0,C 180,E1 21911.327,E2 21911.327} C_VEL
LIN {X 0,Y 479.268,Z 702.044,A -85,B 0,C 180,E1 21907.709,E2 21907.709} C_VEL
LIN {X 0,Y 477.987,Z 760.957,A -85,B 0,C 180,E1 21906.719,E2 21906.719} C_VEL
LIN {X 0,Y 476.86,Z 782.231,A -85,B 0,C 180,E1 21906.16,E2 21906.16} C_VEL
LIN {X 0,Y 475.376,Z 803.883,A -85,B 0,C 180,E1 21905.377,E2 21905.377} C_VEL
LIN {X 0,Y 473.726,Z 823.948,A -85,B 0,C 180,E1 21904.449,E2 21904.449} C_VEL
LIN {X 0,Y 471.815,Z 843.848,A -85,B 0,C 180,E1 21903.291,E2 21903.291} C_VEL
LIN {X 0,Y 469.627,Z 864.445,A -85,B 0,C 180,E1 21901.844,E2 21901.844} C_VEL
LIN {X 0,Y 467.586,Z 882.839,A -85,B 0,C 180,E1 21900.31,E2 21900.31} C_VEL
LIN {X 0,Y 465.442,Z 900.934,A -85,B 0,C 180,E1 21898.526,E2 21898.526} C_VEL
LIN {X 0,Y 463.473,Z 917.681,A -85,B 0,C 180,E1 21896.595,E2 21896.595} C_VEL
LIN {X 0,Y 461.714,Z 932.973,A -85,B 0,C 180,E1 21894.561,E2 21894.561} C_VEL
LIN {X 0,Y 460.293,Z 945.594,A -85,B 0,C 180,E1 21892.603,E2 21892.603} C_VEL
LIN {X 0,Y 458.788,Z 959.262,A -85,B 0,C 180,E1 21890.067,E2 21890.067} C_VEL
LIN {X 0,Y 457.746,Z 970.219,A -85,B 0,C 180,E1 21887.677,E2 21887.677} C_VEL
LIN {X 0,Y 456.935,Z 980.042,A -85,B 0,C 180,E1 21885.096,E2 21885.096} C_VEL
LIN {X 0,Y 456.391,Z 988.461,A -85,B 0,C 180,E1 21882.4,E2 21882.4} C_VEL
LIN {X 0,Y 456.102,Z 994.867,A -85,B 0,C 180,E1 21879.848,E2 21879.848} C_VEL
LIN {X 0,Y 455.959,Z 999.602,A -85,B 0,C 180,E1 21877.309,E2 21877.309} C_VEL
LIN {X 0,Y 455.915,Z 1003.102,A -85,B 0,C 180,E1 21874.657,E2 21874.657} C_VEL
LIN {X 0,Y 455.909,Z 1004.948,A -85,B 0,C 180,E1 21872.139,E2 21872.139} C_VEL
LIN {X 0,Y 455.893,Z 1005.394,A -85,B 0,C 180,E1 21869.374,E2 21869.374} C_VEL
LIN {X 0,Y 455.907,Z 1004.335,A -85,B 0,C 180,E1 21866.734,E2 21866.734} C_VEL
LIN {X 0,Y 455.941,Z 1001.62,A -85,B 0,C 180,E1 21864.087,E2 21864.087} C_VEL
LIN {X 0,Y 456.038,Z 997.166,A -85,B 0,C 180,E1 21861.302,E2 21861.302} C_VEL
LIN {X 0,Y 456.265,Z 991.256,A -85,B 0,C 180,E1 21858.628,E2 21858.628} C_VEL
LIN {X 0,Y 456.668,Z 983.889,A -85,B 0,C 180,E1 21856.067,E2 21856.067} C_VEL
LIN {X 0,Y 457.37,Z 974.361,A -85,B 0,C 180,E1 21853.362,E2 21853.362} C_VEL
LIN {X 0,Y 458.364,Z 963.611,A -85,B 0,C 180,E1 21850.826,E2 21850.826} C_VEL
LIN {X 0,Y 459.632,Z 951.472,A -85,B 0,C 180,E1 21848.434,E2 21848.434} C_VEL
LIN {X 0,Y 461.02,Z 939.082,A -85,B 0,C 180,E1 21846.349,E2 21846.349} C_VEL
LIN {X 0,Y 462.748,Z 923.826,A -85,B 0,C 180,E1 21844.194,E2 21844.194} C_VEL
LIN {X 0,Y 464.611,Z 907.628,A -85,B 0,C 180,E1 21842.234,E2 21842.234} C_VEL
LIN {X 0,Y 466.702,Z 889.457,A -85,B 0,C 180,E1 21840.341,E2 21840.341} C_VEL
LIN {X 0,Y 468.9,Z 870.386,A -85,B 0,C 180,E1 21838.652,E2 21838.652} C_VEL
LIN {X 0,Y 470.902,Z 851.106,A -85,B 0,C 180,E1 21837.223,E2 21837.223} C_VEL
LIN {X 0,Y 472.981,Z 830.143,A -85,B 0,C 180,E1 21835.935,E2 21835.935} C_VEL
LIN {X 0,Y 474.738,Z 809.646,A -85,B 0,C 180,E1 21834.907,E2 21834.907} C_VEL
LIN {X 0,Y 476.263,Z 788.288,A -85,B 0,C 180,E1 21834.075,E2 21834.075} C_VEL
LIN {X 0,Y 477.479,Z 766.787,A -85,B 0,C 180,E1 21833.462,E2 21833.462} C_VEL
LIN {X 0,Y 478.277,Z 742.848,A -85,B 0,C 180,E1 21832.997,E2 21832.997} C_VEL
LIN {X 0,Y 482.663,Z 512.984,A -85,B 0,C 180,E1 21829.235,E2 21829.235} C_VEL
LIN {X 0,Y 483.15,Z 480.92,A -85,B 0,C 180,E1 21828.678,E2 21828.678} C_VEL
LIN {X 0,Y 479.521,Z 457.443,A -85,B 0,C 180,E1 21827.883,E2 21827.883} C_VEL
LIN {X 0,Y 477.766,Z 454.358,A -85,B 0,C 180,E1 21827.625,E2 21827.625} C_VEL
LIN {X 0,Y 469.831,Z 435.827,A -85,B 0,C 180,E1 21825.224,E2 21825.224} C_VEL
LIN {X 0,Y 462.819,Z 421.04,A -85,B 0,C 180,E1 21823.053,E2 21823.053} C_VEL
LIN {X 0,Y 458.557,Z 412.555,A -85,B 0,C 180,E1 21821.685,E2 21821.685} C_VEL
LIN {X 0,Y 457.071,Z 409.045,A -85,B 0,C 180,E1 21821.063,E2 21821.063} C_VEL
LIN {X 0,Y 457.069,Z 408.8,A -85,B 0,C 180,E1 21817.771,E2 21817.771} C_VEL
LIN {X 0,Y 457.07,Z 408.796,A -85,B 0,C 180,E1 21814.056,E2 21814.056} C_VEL
LIN {X 0,Y 457.033,Z 408.806,A -85,B 0,C 180,E1 21810.471,E2 21810.471} C_VEL
LIN {X 0,Y 457.016,Z 408.799,A -85,B 0,C 180,E1 21806.928,E2 21806.928} C_VEL
LIN {X 0,Y 457.038,Z 408.8,A -85,B 0,C 180,E1 21803.326,E2 21803.326} C_VEL
LIN {X 0,Y 457.046,Z 408.801,A -85,B 0,C 180,E1 21799.821,E2 21799.821} C_VEL
LIN {X 0,Y 457.001,Z 408.808,A -85,B 0,C 180,E1 21796.263,E2 21796.263} C_VEL
LIN {X 0,Y 456.996,Z 408.807,A -85,B 0,C 180,E1 21792.509,E2 21792.509} C_VEL
LIN {X 0,Y 457.026,Z 408.798,A -85,B 0,C 180,E1 21788.936,E2 21788.936} C_VEL
LIN {X 0,Y 457.058,Z 408.795,A -85,B 0,C 180,E1 21785.397,E2 21785.397} C_VEL
LIN {X 0,Y 457.028,Z 408.798,A -85,B 0,C 180,E1 21781.755,E2 21781.755} C_VEL
LIN {X 0,Y 457.021,Z 408.804,A -85,B 0,C 180,E1 21778.119,E2 21778.119} C_VEL
LIN {X 0,Y 457.04,Z 408.803,A -85,B 0,C 180,E1 21774.453,E2 21774.453} C_VEL
LIN {X 0,Y 457.076,Z 408.795,A -85,B 0,C 180,E1 21770.938,E2 21770.938} C_VEL
LIN {X 0,Y 457.062,Z 408.803,A -85,B 0,C 180,E1 21767.235,E2 21767.235} C_VEL
LIN {X 0,Y 457.044,Z 408.804,A -85,B 0,C 180,E1 21763.608,E2 21763.608} C_VEL
LIN {X 0,Y 457.101,Z 409.056,A -85,B 0,C 180,E1 21761.177,E2 21761.177} C_VEL
LIN {X 0,Y 458.553,Z 412.532,A -85,B 0,C 180,E1 21760.512,E2 21760.512} C_VEL
LIN {X 0,Y 464.522,Z 425.447,A -85,B 0,C 180,E1 21758.27,E2 21758.27} C_VEL
LIN {X 0,Y 471.431,Z 441.818,A -85,B 0,C 180,E1 21755.703,E2 21755.703} C_VEL
LIN {X 0,Y 475.656,Z 453.001,A -85,B 0,C 180,E1 21754.131,E2 21754.131} C_VEL
LIN {X 0,Y 480.389,Z 479.889,A -85,B 0,C 180,E1 21753.106,E2 21753.106} C_VEL
LIN {X 0,Y 474.566,Z 718.398,A -85,B 0,C 180,E1 21749.029,E2 21749.029} C_VEL
LIN {X 0,Y 473.538,Z 739.31,A -85,B 0,C 180,E1 21748.448,E2 21748.448} C_VEL
LIN {X 0,Y 472.252,Z 759.03,A -85,B 0,C 180,E1 21747.676,E2 21747.676} C_VEL
LIN {X 0,Y 470.663,Z 778.533,A -85,B 0,C 180,E1 21746.684,E2 21746.684} C_VEL
LIN {X 0,Y 469.765,Z 788.444,A -85,B 0,C 180,E1 21746.082,E2 21746.082} C_VEL
LIN {X 0,Y 468.239,Z 795.419,A -85,B 0,C 180,E1 21745.688,E2 21745.688} C_VEL
LIN {X 0,Y 461.164,Z 812.712,A -85,B 0,C 180,E1 21744.768,E2 21744.768} C_VEL
LIN {X 0,Y 459.537,Z 819.079,A -85,B 0,C 180,E1 21744.275,E2 21744.275} C_VEL
LIN {X 0,Y 457.422,Z 836.237,A -85,B 0,C 180,E1 21742.578,E2 21742.578} C_VEL
LIN {X 0,Y 455.476,Z 851.469,A -85,B 0,C 180,E1 21740.786,E2 21740.786} C_VEL
LIN {X 0,Y 453.589,Z 866.168,A -85,B 0,C 180,E1 21738.73,E2 21738.73} C_VEL
LIN {X 0,Y 451.93,Z 879.39,A -85,B 0,C 180,E1 21736.519,E2 21736.519} C_VEL
LIN {X 0,Y 450.564,Z 891.104,A -85,B 0,C 180,E1 21734.166,E2 21734.166} C_VEL
LIN {X 0,Y 449.565,Z 900.719,A -85,B 0,C 180,E1 21731.835,E2 21731.835} C_VEL
LIN {X 0,Y 448.813,Z 909.434,A -85,B 0,C 180,E1 21729.244,E2 21729.244} C_VEL
LIN {X 0,Y 448.351,Z 916.402,A -85,B 0,C 180,E1 21726.598,E2 21726.598} C_VEL
LIN {X 0,Y 448.123,Z 921.421,A -85,B 0,C 180,E1 21724.054,E2 21724.054} C_VEL
LIN {X 0,Y 448.022,Z 924.888,A -85,B 0,C 180,E1 21721.477,E2 21721.477} C_VEL
LIN {X 0,Y 447.987,Z 926.792,A -85,B 0,C 180,E1 21718.818,E2 21718.818} C_VEL
LIN {X 0,Y 447.977,Z 927.098,A -85,B 0,C 180,E1 21716.201,E2 21716.201} C_VEL
LIN {X 0,Y 447.986,Z 925.817,A -85,B 0,C 180,E1 21713.544,E2 21713.544} C_VEL
LIN {X 0,Y 448.063,Z 923.16,A -85,B 0,C 180,E1 21711.052,E2 21711.052} C_VEL
LIN {X 0,Y 448.239,Z 918.494,A -85,B 0,C 180,E1 21708.328,E2 21708.328} C_VEL
LIN {X 0,Y 448.564,Z 912.408,A -85,B 0,C 180,E1 21705.776,E2 21705.776} C_VEL
LIN {X 0,Y 449.151,Z 904.668,A -85,B 0,C 180,E1 21703.252,E2 21703.252} C_VEL
LIN {X 0,Y 450.033,Z 895.136,A -85,B 0,C 180,E1 21700.753,E2 21700.753} C_VEL
LIN {X 0,Y 451.209,Z 884.26,A -85,B 0,C 180,E1 21698.407,E2 21698.407} C_VEL
LIN {X 0,Y 452.658,Z 872.09,A -85,B 0,C 180,E1 21696.211,E2 21696.211} C_VEL
LIN {X 0,Y 454.46,Z 857.663,A -85,B 0,C 180,E1 21694.034,E2 21694.034} C_VEL
LIN {X 0,Y 456.429,Z 842.056,A -85,B 0,C 180,E1 21692.069,E2 21692.069} C_VEL
LIN {X 0,Y 458.396,Z 825.999,A -85,B 0,C 180,E1 21690.372,E2 21690.372} C_VEL
LIN {X 0,Y 460.432,Z 808.408,A -85,B 0,C 180,E1 21688.815,E2 21688.815} C_VEL
LIN {X 0,Y 462.436,Z 789.759,A -85,B 0,C 180,E1 21687.457,E2 21687.457} C_VEL
LIN {X 0,Y 464.179,Z 771.139,A -85,B 0,C 180,E1 21686.354,E2 21686.354} C_VEL
LIN {X 0,Y 465.714,Z 751.639,A -85,B 0,C 180,E1 21685.441,E2 21685.441} C_VEL
LIN {X 0,Y 466.954,Z 731.273,A -85,B 0,C 180,E1 21684.735,E2 21684.735} C_VEL
LIN {X 0,Y 467.782,Z 710.784,A -85,B 0,C 180,E1 21684.247,E2 21684.247} C_VEL
LIN {X 0,Y 473.199,Z 480.169,A -85,B 0,C 180,E1 21680.335,E2 21680.335} C_VEL
LIN {X 0,Y 468.524,Z 455.365,A -85,B 0,C 180,E1 21679.385,E2 21679.385} C_VEL
LIN {X 0,Y 466.708,Z 451.817,A -85,B 0,C 180,E1 21679.068,E2 21679.068} C_VEL
LIN {X 0,Y 459.117,Z 432.631,A -85,B 0,C 180,E1 21676.239,E2 21676.239} C_VEL
LIN {X 0,Y 452.131,Z 417.001,A -85,B 0,C 180,E1 21673.687,E2 21673.687} C_VEL
LIN {X 0,Y 449.17,Z 410.065,A -85,B 0,C 180,E1 21672.476,E2 21672.476} C_VEL
LIN {X 0,Y 449.13,Z 409.768,A -85,B 0,C 180,E1 21670.896,E2 21670.896} C_VEL
LIN {X 0,Y 449.131,Z 409.737,A -85,B 0,C 180,E1 21667.169,E2 21667.169} C_VEL
LIN {X 0,Y 449.124,Z 409.788,A -85,B 0,C 180,E1 21663.416,E2 21663.416} C_VEL
LIN {X 0,Y 449.119,Z 409.781,A -85,B 0,C 180,E1 21659.643,E2 21659.643} C_VEL
LIN {X 0,Y 449.127,Z 409.779,A -85,B 0,C 180,E1 21655.872,E2 21655.872} C_VEL
LIN {X 0,Y 449.133,Z 409.782,A -85,B 0,C 180,E1 21652.087,E2 21652.087} C_VEL
LIN {X 0,Y 449.132,Z 409.788,A -85,B 0,C 180,E1 21648.267,E2 21648.267} C_VEL
LIN {X 0,Y 449.132,Z 409.786,A -85,B 0,C 180,E1 21644.528,E2 21644.528} C_VEL
LIN {X 0,Y 449.122,Z 409.78,A -85,B 0,C 180,E1 21640.804,E2 21640.804} C_VEL
LIN {X 0,Y 449.126,Z 409.772,A -85,B 0,C 180,E1 21637.108,E2 21637.108} C_VEL
LIN {X 0,Y 449.131,Z 409.79,A -85,B 0,C 180,E1 21633.359,E2 21633.359} C_VEL
LIN {X 0,Y 449.127,Z 409.782,A -85,B 0,C 180,E1 21629.619,E2 21629.619} C_VEL
LIN {X 0,Y 449.13,Z 409.766,A -85,B 0,C 180,E1 21625.871,E2 21625.871} C_VEL
LIN {X 0,Y 449.125,Z 409.783,A -85,B 0,C 180,E1 21622.101,E2 21622.101} C_VEL
LIN {X 0,Y 449.128,Z 409.787,A -85,B 0,C 180,E1 21618.295,E2 21618.295} C_VEL
LIN {X 0,Y 449.134,Z 409.77,A -85,B 0,C 180,E1 21614.57,E2 21614.57} C_VEL
LIN {X 0,Y 449.127,Z 409.79,A -85,B 0,C 180,E1 21610.778,E2 21610.778} C_VEL
LIN {X 0,Y 449.13,Z 409.782,A -85,B 0,C 180,E1 21607.033,E2 21607.033} C_VEL
LIN {X 0,Y 449.127,Z 409.766,A -85,B 0,C 180,E1 21603.319,E2 21603.319} C_VEL
LIN {X 0,Y 449.128,Z 409.783,A -85,B 0,C 180,E1 21599.618,E2 21599.618} C_VEL
LIN {X 0,Y 449.131,Z 409.788,A -85,B 0,C 180,E1 21595.834,E2 21595.834} C_VEL
LIN {X 0,Y 449.12,Z 409.772,A -85,B 0,C 180,E1 21592.067,E2 21592.067} C_VEL
LIN {X 0,Y 449.124,Z 409.776,A -85,B 0,C 180,E1 21588.312,E2 21588.312} C_VEL
LIN {X 0,Y 449.136,Z 409.783,A -85,B 0,C 180,E1 21584.57,E2 21584.57} C_VEL
LIN {X 0,Y 449.131,Z 409.787,A -85,B 0,C 180,E1 21580.763,E2 21580.763} C_VEL
LIN {X 0,Y 449.137,Z 409.79,A -85,B 0,C 180,E1 21576.933,E2 21576.933} C_VEL
LIN {X 0,Y 449.13,Z 409.793,A -85,B 0,C 180,E1 21573.133,E2 21573.133} C_VEL
LIN {X 0,Y 449.121,Z 409.792,A -85,B 0,C 180,E1 21569.495,E2 21569.495} C_VEL
LIN {X 0,Y 449.127,Z 409.785,A -85,B 0,C 180,E1 21565.721,E2 21565.721} C_VEL
LIN {X 0,Y 449.134,Z 409.779,A -85,B 0,C 180,E1 21561.928,E2 21561.928} C_VEL
LIN {X 0,Y 449.167,Z 410.009,A -85,B 0,C 180,E1 21559.867,E2 21559.867} C_VEL
LIN {X 0,Y 450.584,Z 413.493,A -85,B 0,C 180,E1 21559.278,E2 21559.278} C_VEL
LIN {X 0,Y 457.691,Z 427.581,A -85,B 0,C 180,E1 21557.033,E2 21557.033} C_VEL
LIN {X 0,Y 466.954,Z 447.636,A -85,B 0,C 180,E1 21554.167,E2 21554.167} C_VEL
LIN {X 0,Y 470.455,Z 455.531,A -85,B 0,C 180,E1 21553.177,E2 21553.177} C_VEL
LIN {X 0,Y 474.371,Z 462.623,A -85,B 0,C 180,E1 21552.631,E2 21552.631} C_VEL
LIN {X 0,Y 477.43,Z 484.619,A -85,B 0,C 180,E1 21551.905,E2 21551.905} C_VEL
LIN {X 0,Y 472.701,Z 703.927,A -85,B 0,C 180,E1 21548.237,E2 21548.237} C_VEL
LIN {X 0,Y 471.38,Z 760.593,A -85,B 0,C 180,E1 21547.273,E2 21547.273} C_VEL
LIN {X 0,Y 470.174,Z 782.106,A -85,B 0,C 180,E1 21546.702,E2 21546.702} C_VEL
LIN {X 0,Y 468.575,Z 804.026,A -85,B 0,C 180,E1 21545.896,E2 21545.896} C_VEL
LIN {X 0,Y 466.805,Z 824.137,A -85,B 0,C 180,E1 21544.948,E2 21544.948} C_VEL
LIN {X 0,Y 464.802,Z 843.798,A -85,B 0,C 180,E1 21543.787,E2 21543.787} C_VEL
LIN {X 0,Y 462.517,Z 863.972,A -85,B 0,C 180,E1 21542.349,E2 21542.349} C_VEL
LIN {X 0,Y 460.316,Z 882.504,A -85,B 0,C 180,E1 21540.78,E2 21540.78} C_VEL
LIN {X 0,Y 458.07,Z 900.415,A -85,B 0,C 180,E1 21538.987,E2 21538.987} C_VEL
LIN {X 0,Y 455.936,Z 917.365,A -85,B 0,C 180,E1 21536.999,E2 21536.999} C_VEL
LIN {X 0,Y 453.989,Z 933.129,A -85,B 0,C 180,E1 21534.855,E2 21534.855} C_VEL
LIN {X 0,Y 452.339,Z 947.224,A -85,B 0,C 180,E1 21532.622,E2 21532.622} C_VEL
LIN {X 0,Y 450.942,Z 960.079,A -85,B 0,C 180,E1 21530.239,E2 21530.239} C_VEL
LIN {X 0,Y 449.917,Z 970.266,A -85,B 0,C 180,E1 21527.984,E2 21527.984} C_VEL
LIN {X 0,Y 449.039,Z 980.041,A -85,B 0,C 180,E1 21525.368,E2 21525.368} C_VEL
LIN {X 0,Y 448.446,Z 988.461,A -85,B 0,C 180,E1 21522.623,E2 21522.623} C_VEL
LIN {X 0,Y 448.125,Z 994.867,A -85,B 0,C 180,E1 21520.025,E2 21520.025} C_VEL
LIN {X 0,Y 447.965,Z 999.602,A -85,B 0,C 180,E1 21517.441,E2 21517.441} C_VEL
LIN {X 0,Y 447.913,Z 1003.101,A -85,B 0,C 180,E1 21514.74,E2 21514.74} C_VEL
LIN {X 0,Y 447.908,Z 1004.948,A -85,B 0,C 180,E1 21512.177,E2 21512.177} C_VEL
LIN {X 0,Y 447.894,Z 1005.394,A -85,B 0,C 180,E1 21509.363,E2 21509.363} C_VEL
LIN {X 0,Y 447.909,Z 1004.335,A -85,B 0,C 180,E1 21506.676,E2 21506.676} C_VEL
LIN {X 0,Y 447.944,Z 1001.619,A -85,B 0,C 180,E1 21503.981,E2 21503.981} C_VEL
LIN {X 0,Y 448.05,Z 997.166,A -85,B 0,C 180,E1 21501.145,E2 21501.145} C_VEL
LIN {X 0,Y 448.302,Z 991.256,A -85,B 0,C 180,E1 21498.424,E2 21498.424} C_VEL
LIN {X 0,Y 448.757,Z 983.664,A -85,B 0,C 180,E1 21495.743,E2 21495.743} C_VEL
LIN {X 0,Y 449.551,Z 973.845,A -85,B 0,C 180,E1 21492.931,E2 21492.931} C_VEL
LIN {X 0,Y 450.618,Z 963.361,A -85,B 0,C 180,E1 21490.428,E2 21490.428} C_VEL
LIN {X 0,Y 451.828,Z 951.704,A -85,B 0,C 180,E1 21488.179,E2 21488.179} C_VEL
LIN {X 0,Y 453.468,Z 937.286,A -85,B 0,C 180,E1 21485.792,E2 21485.792} C_VEL
LIN {X 0,Y 455.299,Z 922.155,A -85,B 0,C 180,E1 21483.635,E2 21483.635} C_VEL
LIN {X 0,Y 457.341,Z 905.52,A -85,B 0,C 180,E1 21481.617,E2 21481.617} C_VEL
LIN {X 0,Y 459.623,Z 887.006,A -85,B 0,C 180,E1 21479.693,E2 21479.693} C_VEL
LIN {X 0,Y 461.831,Z 868.656,A -85,B 0,C 180,E1 21478.067,E2 21478.067} C_VEL
LIN {X 0,Y 463.927,Z 849.885,A -85,B 0,C 180,E1 21476.666,E2 21476.666} C_VEL
LIN {X 0,Y 466.013,Z 829.926,A -85,B 0,C 180,E1 21475.428,E2 21475.428} C_VEL
LIN {X 0,Y 467.879,Z 809.539,A -85,B 0,C 180,E1 21474.39,E2 21474.39} C_VEL
LIN {X 0,Y 469.504,Z 788.176,A -85,B 0,C 180,E1 21473.547,E2 21473.547} C_VEL
LIN {X 0,Y 470.81,Z 766.464,A -85,B 0,C 180,E1 21472.919,E2 21472.919} C_VEL
LIN {X 0,Y 471.651,Z 742.748,A -85,B 0,C 180,E1 21472.452,E2 21472.452} C_VEL
LIN {X 0,Y 476.324,Z 514.915,A -85,B 0,C 180,E1 21468.675,E2 21468.675} C_VEL
LIN {X 0,Y 476.866,Z 482.322,A -85,B 0,C 180,E1 21468.102,E2 21468.102} C_VEL
LIN {X 0,Y 473.69,Z 461.406,A -85,B 0,C 180,E1 21467.381,E2 21467.381} C_VEL
LIN {X 0,Y 469.684,Z 454.437,A -85,B 0,C 180,E1 21466.811,E2 21466.811} C_VEL
LIN {X 0,Y 461.876,Z 436.487,A -85,B 0,C 180,E1 21464.364,E2 21464.364} C_VEL
LIN {X 0,Y 455.266,Z 422.52,A -85,B 0,C 180,E1 21462.224,E2 21462.224} C_VEL
LIN {X 0,Y 450.693,Z 413.672,A -85,B 0,C 180,E1 21460.71,E2 21460.71} C_VEL
LIN {X 0,Y 449.173,Z 410.019,A -85,B 0,C 180,E1 21460.033,E2 21460.033} C_VEL
LIN {X 0,Y 449.111,Z 409.787,A -85,B 0,C 180,E1 21456.471,E2 21456.471} C_VEL
LIN {X 0,Y 449.089,Z 409.796,A -85,B 0,C 180,E1 21452.904,E2 21452.904} C_VEL
LIN {X 0,Y 449.089,Z 409.789,A -85,B 0,C 180,E1 21449.182,E2 21449.182} C_VEL
LIN {X 0,Y 449.12,Z 409.79,A -85,B 0,C 180,E1 21445.587,E2 21445.587} C_VEL
LIN {X 0,Y 449.102,Z 409.794,A -85,B 0,C 180,E1 21441.964,E2 21441.964} C_VEL
LIN {X 0,Y 449.063,Z 409.793,A -85,B 0,C 180,E1 21438.431,E2 21438.431} C_VEL
LIN {X 0,Y 449.056,Z 409.788,A -85,B 0,C 180,E1 21434.704,E2 21434.704} C_VEL
LIN {X 0,Y 449.098,Z 409.786,A -85,B 0,C 180,E1 21431.168,E2 21431.168} C_VEL
LIN {X 0,Y 449.122,Z 409.786,A -85,B 0,C 180,E1 21427.419,E2 21427.419} C_VEL
LIN {X 0,Y 449.092,Z 409.795,A -85,B 0,C 180,E1 21423.702,E2 21423.702} C_VEL
LIN {X 0,Y 449.08,Z 409.795,A -85,B 0,C 180,E1 21420.127,E2 21420.127} C_VEL
LIN {X 0,Y 449.095,Z 409.785,A -85,B 0,C 180,E1 21416.426,E2 21416.426} C_VEL
LIN {X 0,Y 449.139,Z 409.787,A -85,B 0,C 180,E1 21412.838,E2 21412.838} C_VEL
LIN {X 0,Y 449.132,Z 409.786,A -85,B 0,C 180,E1 21409.092,E2 21409.092} C_VEL
LIN {X 0,Y 449.113,Z 409.794,A -85,B 0,C 180,E1 21405.429,E2 21405.429} C_VEL
LIN {X 0,Y 449.158,Z 410.04,A -85,B 0,C 180,E1 21402.21,E2 21402.21} C_VEL
LIN {X 0,Y 450.644,Z 413.601,A -85,B 0,C 180,E1 21401.501,E2 21401.501} C_VEL
LIN {X 0,Y 455.584,Z 424.078,A -85,B 0,C 180,E1 21399.576,E2 21399.576} C_VEL
LIN {X 0,Y 462.454,Z 439.749,A -85,B 0,C 180,E1 21396.962,E2 21396.962} C_VEL
LIN {X 0,Y 467.88,Z 453.298,A -85,B 0,C 180,E1 21394.952,E2 21394.952} C_VEL
LIN {X 0,Y 470.087,Z 457.532,A -85,B 0,C 180,E1 21394.622,E2 21394.622} C_VEL
LIN {X 0,Y 474.189,Z 481.43,A -85,B 0,C 180,E1 21393.696,E2 21393.696} C_VEL
LIN {X 0,Y 467.971,Z 719.054,A -85,B 0,C 180,E1 21389.574,E2 21389.574} C_VEL
LIN {X 0,Y 466.879,Z 740.117,A -85,B 0,C 180,E1 21388.98,E2 21388.98} C_VEL
LIN {X 0,Y 465.493,Z 760.103,A -85,B 0,C 180,E1 21388.182,E2 21388.182} C_VEL
LIN {X 0,Y 463.852,Z 779.041,A -85,B 0,C 180,E1 21387.203,E2 21387.203} C_VEL
LIN {X 0,Y 461.96,Z 797.893,A -85,B 0,C 180,E1 21385.984,E2 21385.984} C_VEL
LIN {X 0,Y 459.984,Z 815.543,A -85,B 0,C 180,E1 21384.593,E2 21384.593} C_VEL
LIN {X 0,Y 459.537,Z 819.079,A -85,B 0,C 180,E1 21384.275,E2 21384.275} C_VEL
LIN {X 0,Y 457.896,Z 825.483,A -85,B 0,C 180,E1 21383.75,E2 21383.75} C_VEL
LIN {X 0,Y 450.546,Z 841.299,A -85,B 0,C 180,E1 21382.485,E2 21382.485} C_VEL
LIN {X 0,Y 448.861,Z 847.009,A -85,B 0,C 180,E1 21381.866,E2 21381.866} C_VEL
LIN {X 0,Y 446.814,Z 861.875,A -85,B 0,C 180,E1 21379.873,E2 21379.873} C_VEL
LIN {X 0,Y 445.026,Z 874.983,A -85,B 0,C 180,E1 21377.795,E2 21377.795} C_VEL
LIN {X 0,Y 443.445,Z 887.278,A -85,B 0,C 180,E1 21375.474,E2 21375.474} C_VEL
LIN {X 0,Y 442.154,Z 898.193,A -85,B 0,C 180,E1 21372.979,E2 21372.979} C_VEL
LIN {X 0,Y 441.224,Z 907.381,A -85,B 0,C 180,E1 21370.394,E2 21370.394} C_VEL
LIN {X 0,Y 440.617,Z 914.609,A -85,B 0,C 180,E1 21367.843,E2 21367.843} C_VEL
LIN {X 0,Y 440.269,Z 920.44,A -85,B 0,C 180,E1 21365.157,E2 21365.157} C_VEL
LIN {X 0,Y 440.081,Z 924.624,A -85,B 0,C 180,E1 21362.42,E2 21362.42} C_VEL
LIN {X 0,Y 440.03,Z 927.065,A -85,B 0,C 180,E1 21359.772,E2 21359.772} C_VEL
LIN {X 0,Y 440.01,Z 927.932,A -85,B 0,C 180,E1 21357.03,E2 21357.03} C_VEL
LIN {X 0,Y 440.02,Z 927.113,A -85,B 0,C 180,E1 21354.328,E2 21354.328} C_VEL
LIN {X 0,Y 440.066,Z 924.746,A -85,B 0,C 180,E1 21351.677,E2 21351.677} C_VEL
LIN {X 0,Y 440.23,Z 920.649,A -85,B 0,C 180,E1 21348.949,E2 21348.949} C_VEL
LIN {X 0,Y 440.541,Z 915.092,A -85,B 0,C 180,E1 21346.342,E2 21346.342} C_VEL
LIN {X 0,Y 441.11,Z 907.899,A -85,B 0,C 180,E1 21343.765,E2 21343.765} C_VEL
LIN {X 0,Y 442.021,Z 898.39,A -85,B 0,C 180,E1 21341.082,E2 21341.082} C_VEL
LIN {X 0,Y 443.199,Z 887.954,A -85,B 0,C 180,E1 21338.691,E2 21338.691} C_VEL
LIN {X 0,Y 444.698,Z 875.887,A -85,B 0,C 180,E1 21336.384,E2 21336.384} C_VEL
LIN {X 0,Y 446.479,Z 862.484,A -85,B 0,C 180,E1 21334.235,E2 21334.235} C_VEL
LIN {X 0,Y 448.467,Z 847.677,A -85,B 0,C 180,E1 21332.233,E2 21332.233} C_VEL
LIN {X 0,Y 450.572,Z 831.95,A -85,B 0,C 180,E1 21330.442,E2 21330.442} C_VEL
LIN {X 0,Y 452.77,Z 814.647,A -85,B 0,C 180,E1 21328.795,E2 21328.795} C_VEL
LIN {X 0,Y 454.792,Z 797.102,A -85,B 0,C 180,E1 21327.414,E2 21327.414} C_VEL
LIN {X 0,Y 456.692,Z 778.823,A -85,B 0,C 180,E1 21326.232,E2 21326.232} C_VEL
LIN {X 0,Y 458.432,Z 759.127,A -85,B 0,C 180,E1 21325.212,E2 21325.212} C_VEL
LIN {X 0,Y 459.87,Z 739.056,A -85,B 0,C 180,E1 21324.418,E2 21324.418} C_VEL
LIN {X 0,Y 460.967,Z 718.27,A -85,B 0,C 180,E1 21323.834,E2 21323.834} C_VEL
LIN {X 0,Y 466.972,Z 481.881,A -85,B 0,C 180,E1 21319.753,E2 21319.753} C_VEL
LIN {X 0,Y 462.735,Z 459.234,A -85,B 0,C 180,E1 21318.866,E2 21318.866} C_VEL
LIN {X 0,Y 458.889,Z 452.498,A -85,B 0,C 180,E1 21318.307,E2 21318.307} C_VEL
LIN {X 0,Y 451.386,Z 433.833,A -85,B 0,C 180,E1 21315.466,E2 21315.466} C_VEL
LIN {X 0,Y 444.208,Z 417.94,A -85,B 0,C 180,E1 21312.774,E2 21312.774} C_VEL
LIN {X 0,Y 441.232,Z 411.069,A -85,B 0,C 180,E1 21311.535,E2 21311.535} C_VEL
LIN {X 0,Y 441.182,Z 410.775,A -85,B 0,C 180,E1 21309.709,E2 21309.709} C_VEL
LIN {X 0,Y 441.177,Z 410.741,A -85,B 0,C 180,E1 21305.922,E2 21305.922} C_VEL
LIN {X 0,Y 441.195,Z 410.768,A -85,B 0,C 180,E1 21302.168,E2 21302.168} C_VEL
LIN {X 0,Y 441.191,Z 410.766,A -85,B 0,C 180,E1 21298.43,E2 21298.43} C_VEL
LIN {X 0,Y 441.192,Z 410.763,A -85,B 0,C 180,E1 21294.673,E2 21294.673} C_VEL
LIN {X 0,Y 441.185,Z 410.76,A -85,B 0,C 180,E1 21290.945,E2 21290.945} C_VEL
LIN {X 0,Y 441.18,Z 410.763,A -85,B 0,C 180,E1 21287.162,E2 21287.162} C_VEL
LIN {X 0,Y 441.188,Z 410.772,A -85,B 0,C 180,E1 21283.323,E2 21283.323} C_VEL
LIN {X 0,Y 441.197,Z 410.776,A -85,B 0,C 180,E1 21279.555,E2 21279.555} C_VEL
LIN {X 0,Y 441.188,Z 410.763,A -85,B 0,C 180,E1 21275.772,E2 21275.772} C_VEL
LIN {X 0,Y 441.194,Z 410.764,A -85,B 0,C 180,E1 21272.026,E2 21272.026} C_VEL
LIN {X 0,Y 441.188,Z 410.776,A -85,B 0,C 180,E1 21268.272,E2 21268.272} C_VEL
LIN {X 0,Y 441.186,Z 410.767,A -85,B 0,C 180,E1 21264.503,E2 21264.503} C_VEL
LIN {X 0,Y 441.192,Z 410.758,A -85,B 0,C 180,E1 21260.704,E2 21260.704} C_VEL
LIN {X 0,Y 441.189,Z 410.78,A -85,B 0,C 180,E1 21256.863,E2 21256.863} C_VEL
LIN {X 0,Y 441.186,Z 410.768,A -85,B 0,C 180,E1 21253.099,E2 21253.099} C_VEL
LIN {X 0,Y 441.192,Z 410.761,A -85,B 0,C 180,E1 21249.391,E2 21249.391} C_VEL
LIN {X 0,Y 441.189,Z 410.775,A -85,B 0,C 180,E1 21245.593,E2 21245.593} C_VEL
LIN {X 0,Y 441.19,Z 410.768,A -85,B 0,C 180,E1 21241.819,E2 21241.819} C_VEL
LIN {X 0,Y 441.187,Z 410.76,A -85,B 0,C 180,E1 21238.052,E2 21238.052} C_VEL
LIN {X 0,Y 441.183,Z 410.776,A -85,B 0,C 180,E1 21234.227,E2 21234.227} C_VEL
LIN {X 0,Y 441.19,Z 410.777,A -85,B 0,C 180,E1 21230.478,E2 21230.478} C_VEL
LIN {X 0,Y 441.196,Z 410.773,A -85,B 0,C 180,E1 21226.635,E2 21226.635} C_VEL
LIN {X 0,Y 441.19,Z 410.765,A -85,B 0,C 180,E1 21222.866,E2 21222.866} C_VEL
LIN {X 0,Y 441.194,Z 410.764,A -85,B 0,C 180,E1 21219.158,E2 21219.158} C_VEL
LIN {X 0,Y 441.18,Z 410.768,A -85,B 0,C 180,E1 21215.498,E2 21215.498} C_VEL
LIN {X 0,Y 441.185,Z 410.767,A -85,B 0,C 180,E1 21211.728,E2 21211.728} C_VEL
LIN {X 0,Y 441.193,Z 410.765,A -85,B 0,C 180,E1 21207.974,E2 21207.974} C_VEL
LIN {X 0,Y 441.193,Z 410.771,A -85,B 0,C 180,E1 21204.219,E2 21204.219} C_VEL
LIN {X 0,Y 441.22,Z 411.035,A -85,B 0,C 180,E1 21200.876,E2 21200.876} C_VEL
LIN {X 0,Y 442.638,Z 414.454,A -85,B 0,C 180,E1 21200.264,E2 21200.264} C_VEL
LIN {X 0,Y 443.796,Z 416.628,A -85,B 0,C 180,E1 21199.884,E2 21199.884} C_VEL
LIN {X 0,Y 451.774,Z 432.56,A -85,B 0,C 180,E1 21197.29,E2 21197.29} C_VEL
LIN {X 0,Y 460.966,Z 452.654,A -85,B 0,C 180,E1 21194.382,E2 21194.382} C_VEL
LIN {X 0,Y 462.783,Z 456.332,A -85,B 0,C 180,E1 21193.968,E2 21193.968} C_VEL
LIN {X 0,Y 468.555,Z 466.415,A -85,B 0,C 180,E1 21193.153,E2 21193.153} C_VEL
LIN {X 0,Y 471.205,Z 486.114,A -85,B 0,C 180,E1 21192.495,E2 21192.495} C_VEL
LIN {X 0,Y 466.169,Z 705.678,A -85,B 0,C 180,E1 21188.782,E2 21188.782} C_VEL
LIN {X 0,Y 464.815,Z 760.29,A -85,B 0,C 180,E1 21187.84,E2 21187.84} C_VEL
LIN {X 0,Y 463.535,Z 781.94,A -85,B 0,C 180,E1 21187.259,E2 21187.259} C_VEL
LIN {X 0,Y 461.875,Z 803.464,A -85,B 0,C 180,E1 21186.46,E2 21186.46} C_VEL
LIN {X 0,Y 459.958,Z 823.988,A -85,B 0,C 180,E1 21185.481,E2 21185.481} C_VEL
LIN {X 0,Y 457.823,Z 843.748,A -85,B 0,C 180,E1 21184.297,E2 21184.297} C_VEL
LIN {X 0,Y 455.405,Z 863.827,A -85,B 0,C 180,E1 21182.842,E2 21182.842} C_VEL
LIN {X 0,Y 452.994,Z 882.8,A -85,B 0,C 180,E1 21181.203,E2 21181.203} C_VEL
LIN {X 0,Y 450.614,Z 900.783,A -85,B 0,C 180,E1 21179.367,E2 21179.367} C_VEL
LIN {X 0,Y 448.349,Z 917.572,A -85,B 0,C 180,E1 21177.35,E2 21177.35} C_VEL
LIN {X 0,Y 446.193,Z 933.929,A -85,B 0,C 180,E1 21175.059,E2 21175.059} C_VEL
LIN {X 0,Y 444.425,Z 948.26,A -85,B 0,C 180,E1 21172.72,E2 21172.72} C_VEL
LIN {X 0,Y 442.932,Z 961.295,A -85,B 0,C 180,E1 21170.207,E2 21170.207} C_VEL
LIN {X 0,Y 441.799,Z 972.523,A -85,B 0,C 180,E1 21167.656,E2 21167.656} C_VEL
LIN {X 0,Y 441.076,Z 980.958,A -85,B 0,C 180,E1 21165.383,E2 21165.383} C_VEL
LIN {X 0,Y 440.479,Z 988.814,A -85,B 0,C 180,E1 21162.722,E2 21162.722} C_VEL
LIN {X 0,Y 440.123,Z 995.378,A -85,B 0,C 180,E1 21159.945,E2 21159.945} C_VEL
LIN {X 0,Y 439.964,Z 1000.014,A -85,B 0,C 180,E1 21157.314,E2 21157.314} C_VEL
LIN {X 0,Y 439.92,Z 1003.442,A -85,B 0,C 180,E1 21154.435,E2 21154.435} C_VEL
LIN {X 0,Y 439.9,Z 1005.208,A -85,B 0,C 180,E1 21151.696,E2 21151.696} C_VEL
LIN {X 0,Y 439.9,Z 1005.348,A -85,B 0,C 180,E1 21149.091,E2 21149.091} C_VEL
LIN {X 0,Y 439.912,Z 1004.125,A -85,B 0,C 180,E1 21146.354,E2 21146.354} C_VEL
LIN {X 0,Y 439.956,Z 1001.299,A -85,B 0,C 180,E1 21143.609,E2 21143.609} C_VEL
LIN {X 0,Y 440.074,Z 996.912,A -85,B 0,C 180,E1 21140.852,E2 21140.852} C_VEL
LIN {X 0,Y 440.358,Z 990.943,A -85,B 0,C 180,E1 21138.079,E2 21138.079} C_VEL
LIN {X 0,Y 440.852,Z 983.483,A -85,B 0,C 180,E1 21135.422,E2 21135.422} C_VEL
LIN {X 0,Y 441.554,Z 975.23,A -85,B 0,C 180,E1 21133.019,E2 21133.019} C_VEL
LIN {X 0,Y 442.597,Z 964.418,A -85,B 0,C 180,E1 21130.471,E2 21130.471} C_VEL
LIN {X 0,Y 443.916,Z 952.295,A -85,B 0,C 180,E1 21128.048,E2 21128.048} C_VEL
LIN {X 0,Y 445.627,Z 938.134,A -85,B 0,C 180,E1 21125.62,E2 21125.62} C_VEL
LIN {X 0,Y 447.563,Z 922.906,A -85,B 0,C 180,E1 21123.394,E2 21123.394} C_VEL
LIN {X 0,Y 449.748,Z 906.21,A -85,B 0,C 180,E1 21121.306,E2 21121.306} C_VEL
LIN {X 0,Y 452.181,Z 887.748,A -85,B 0,C 180,E1 21119.333,E2 21119.333} C_VEL
LIN {X 0,Y 454.588,Z 868.984,A -85,B 0,C 180,E1 21117.629,E2 21117.629} C_VEL
LIN {X 0,Y 456.877,Z 849.683,A -85,B 0,C 180,E1 21116.166,E2 21116.166} C_VEL
LIN {X 0,Y 459.084,Z 829.718,A -85,B 0,C 180,E1 21114.907,E2 21114.907} C_VEL
LIN {X 0,Y 461.065,Z 809.451,A -85,B 0,C 180,E1 21113.858,E2 21113.858} C_VEL
LIN {X 0,Y 462.797,Z 787.98,A -85,B 0,C 180,E1 21113,E2 21113} C_VEL
LIN {X 0,Y 464.192,Z 766.074,A -85,B 0,C 180,E1 21112.358,E2 21112.358} C_VEL
LIN {X 0,Y 465.074,Z 742.513,A -85,B 0,C 180,E1 21111.888,E2 21111.888} C_VEL
LIN {X 0,Y 470.053,Z 515.957,A -85,B 0,C 180,E1 21108.083,E2 21108.083} C_VEL
LIN {X 0,Y 470.626,Z 483.696,A -85,B 0,C 180,E1 21107.509,E2 21107.509} C_VEL
LIN {X 0,Y 467.846,Z 465.201,A -85,B 0,C 180,E1 21106.857,E2 21106.857} C_VEL
LIN {X 0,Y 461.517,Z 454.178,A -85,B 0,C 180,E1 21105.904,E2 21105.904} C_VEL
LIN {X 0,Y 453.477,Z 435.968,A -85,B 0,C 180,E1 21103.291,E2 21103.291} C_VEL
LIN {X 0,Y 446.957,Z 422.833,A -85,B 0,C 180,E1 21101.123,E2 21101.123} C_VEL
LIN {X 0,Y 442.955,Z 414.89,A -85,B 0,C 180,E1 21099.702,E2 21099.702} C_VEL
LIN {X 0,Y 441.239,Z 411.292,A -85,B 0,C 180,E1 21099.012,E2 21099.012} C_VEL
LIN {X 0,Y 441.186,Z 410.775,A -85,B 0,C 180,E1 21098.366,E2 21098.366} C_VEL
LIN {X 0,Y 441.156,Z 410.779,A -85,B 0,C 180,E1 21094.649,E2 21094.649} C_VEL
LIN {X 0,Y 441.146,Z 410.784,A -85,B 0,C 180,E1 21090.963,E2 21090.963} C_VEL
LIN {X 0,Y 441.159,Z 410.777,A -85,B 0,C 180,E1 21087.331,E2 21087.331} C_VEL
LIN {X 0,Y 441.189,Z 410.772,A -85,B 0,C 180,E1 21083.649,E2 21083.649} C_VEL
LIN {X 0,Y 441.151,Z 410.779,A -85,B 0,C 180,E1 21080.013,E2 21080.013} C_VEL
LIN {X 0,Y 441.12,Z 410.787,A -85,B 0,C 180,E1 21076.459,E2 21076.459} C_VEL
LIN {X 0,Y 441.123,Z 410.785,A -85,B 0,C 180,E1 21072.701,E2 21072.701} C_VEL
LIN {X 0,Y 441.166,Z 410.776,A -85,B 0,C 180,E1 21069.128,E2 21069.128} C_VEL
LIN {X 0,Y 441.173,Z 410.773,A -85,B 0,C 180,E1 21065.462,E2 21065.462} C_VEL
LIN {X 0,Y 441.147,Z 410.775,A -85,B 0,C 180,E1 21061.818,E2 21061.818} C_VEL
LIN {X 0,Y 441.144,Z 410.783,A -85,B 0,C 180,E1 21058.102,E2 21058.102} C_VEL
LIN {X 0,Y 441.161,Z 410.781,A -85,B 0,C 180,E1 21054.407,E2 21054.407} C_VEL
LIN {X 0,Y 441.193,Z 410.773,A -85,B 0,C 180,E1 21050.74,E2 21050.74} C_VEL
LIN {X 0,Y 441.195,Z 410.776,A -85,B 0,C 180,E1 21047.01,E2 21047.01} C_VEL
LIN {X 0,Y 441.191,Z 410.905,A -85,B 0,C 180,E1 21043.408,E2 21043.408} C_VEL
LIN {X 0,Y 441.387,Z 411.813,A -85,B 0,C 180,E1 21043.144,E2 21043.144} C_VEL
LIN {X 0,Y 443.707,Z 416.698,A -85,B 0,C 180,E1 21042.153,E2 21042.153} C_VEL
LIN {X 0,Y 447.982,Z 425.63,A -85,B 0,C 180,E1 21040.44,E2 21040.44} C_VEL
LIN {X 0,Y 454.147,Z 439.414,A -85,B 0,C 180,E1 21038.02,E2 21038.02} C_VEL
LIN {X 0,Y 459.836,Z 453.326,A -85,B 0,C 180,E1 21035.854,E2 21035.854} C_VEL
LIN {X 0,Y 464.494,Z 461.625,A -85,B 0,C 180,E1 21035.147,E2 21035.147} C_VEL
LIN {X 0,Y 468.054,Z 483.085,A -85,B 0,C 180,E1 21034.302,E2 21034.302} C_VEL
LIN {X 0,Y 461.431,Z 719.478,A -85,B 0,C 180,E1 21030.14,E2 21030.14} C_VEL
LIN {X 0,Y 460.279,Z 740.613,A -85,B 0,C 180,E1 21029.536,E2 21029.536} C_VEL
LIN {X 0,Y 458.867,Z 759.899,A -85,B 0,C 180,E1 21028.761,E2 21028.761} C_VEL
LIN {X 0,Y 457.096,Z 779.496,A -85,B 0,C 180,E1 21027.742,E2 21027.742} C_VEL
LIN {X 0,Y 455.134,Z 798.009,A -85,B 0,C 180,E1 21026.536,E2 21026.536} C_VEL
LIN {X 0,Y 453.052,Z 815.616,A -85,B 0,C 180,E1 21025.138,E2 21025.138} C_VEL
LIN {X 0,Y 450.796,Z 832.925,A -85,B 0,C 180,E1 21023.475,E2 21023.475} C_VEL
LIN {X 0,Y 448.861,Z 847.009,A -85,B 0,C 180,E1 21021.866,E2 21021.866} C_VEL
LIN {X 0,Y 447.176,Z 852.696,A -85,B 0,C 180,E1 21021.217,E2 21021.217} C_VEL
LIN {X 0,Y 439.739,Z 866.725,A -85,B 0,C 180,E1 21019.612,E2 21019.612} C_VEL
LIN {X 0,Y 438.103,Z 871.655,A -85,B 0,C 180,E1 21018.872,E2 21018.872} C_VEL
LIN {X 0,Y 436.277,Z 884.537,A -85,B 0,C 180,E1 21016.523,E2 21016.523} C_VEL
LIN {X 0,Y 434.755,Z 896.062,A -85,B 0,C 180,E1 21013.985,E2 21013.985} C_VEL
LIN {X 0,Y 433.66,Z 905.586,A -85,B 0,C 180,E1 21011.425,E2 21011.425} C_VEL
LIN {X 0,Y 432.917,Z 913.235,A -85,B 0,C 180,E1 21008.891,E2 21008.891} C_VEL
LIN {X 0,Y 432.436,Z 919.68,A -85,B 0,C 180,E1 21006.124,E2 21006.124} C_VEL
LIN {X 0,Y 432.189,Z 924.286,A -85,B 0,C 180,E1 21003.366,E2 21003.366} C_VEL
LIN {X 0,Y 432.08,Z 927.102,A -85,B 0,C 180,E1 21000.753,E2 21000.753} C_VEL
LIN {X 0,Y 432.044,Z 928.504,A -85,B 0,C 180,E1 20998.017,E2 20998.017} C_VEL
LIN {X 0,Y 432.043,Z 928.357,A -85,B 0,C 180,E1 20995.345,E2 20995.345} C_VEL
LIN {X 0,Y 432.091,Z 926.544,A -85,B 0,C 180,E1 20992.586,E2 20992.586} C_VEL
LIN {X 0,Y 432.208,Z 923.145,A -85,B 0,C 180,E1 20989.877,E2 20989.877} C_VEL
LIN {X 0,Y 432.473,Z 918.2,A -85,B 0,C 180,E1 20987.21,E2 20987.21} C_VEL
LIN {X 0,Y 432.974,Z 911.668,A -85,B 0,C 180,E1 20984.575,E2 20984.575} C_VEL
LIN {X 0,Y 433.779,Z 903.446,A -85,B 0,C 180,E1 20981.97,E2 20981.97} C_VEL
LIN {X 0,Y 434.953,Z 893.344,A -85,B 0,C 180,E1 20979.39,E2 20979.39} C_VEL
LIN {X 0,Y 436.444,Z 881.795,A -85,B 0,C 180,E1 20976.971,E2 20976.971} C_VEL
LIN {X 0,Y 438.235,Z 868.862,A -85,B 0,C 180,E1 20974.708,E2 20974.708} C_VEL
LIN {X 0,Y 440.288,Z 854.527,A -85,B 0,C 180,E1 20972.6,E2 20972.6} C_VEL
LIN {X 0,Y 442.541,Z 838.696,A -85,B 0,C 180,E1 20970.644,E2 20970.644} C_VEL
LIN {X 0,Y 444.767,Z 822.539,A -85,B 0,C 180,E1 20968.967,E2 20968.967} C_VEL
LIN {X 0,Y 447.046,Z 804.856,A -85,B 0,C 180,E1 20967.434,E2 20967.434} C_VEL
LIN {X 0,Y 449.2,Z 786.071,A -85,B 0,C 180,E1 20966.105,E2 20966.105} C_VEL
LIN {X 0,Y 451.048,Z 767.342,A -85,B 0,C 180,E1 20965.038,E2 20965.038} C_VEL
LIN {X 0,Y 452.72,Z 746.83,A -85,B 0,C 180,E1 20964.127,E2 20964.127} C_VEL
LIN {X 0,Y 454.004,Z 725.924,A -85,B 0,C 180,E1 20963.449,E2 20963.449} C_VEL
LIN {X 0,Y 454.861,Z 703.848,A -85,B 0,C 180,E1 20962.978,E2 20962.978} C_VEL
LIN {X 0,Y 460.697,Z 483.09,A -85,B 0,C 180,E1 20959.138,E2 20959.138} C_VEL
LIN {X 0,Y 457.103,Z 463.338,A -85,B 0,C 180,E1 20958.352,E2 20958.352} C_VEL
LIN {X 0,Y 450.77,Z 452.461,A -85,B 0,C 180,E1 20957.415,E2 20957.415} C_VEL
LIN {X 0,Y 443.708,Z 435.154,A -85,B 0,C 180,E1 20954.681,E2 20954.681} C_VEL
LIN {X 0,Y 436.526,Z 419.353,A -85,B 0,C 180,E1 20951.908,E2 20951.908} C_VEL
LIN {X 0,Y 433.291,Z 412.009,A -85,B 0,C 180,E1 20950.52,E2 20950.52} C_VEL
LIN {X 0,Y 433.25,Z 411.712,A -85,B 0,C 180,E1 20946.898,E2 20946.898} C_VEL
LIN {X 0,Y 433.254,Z 411.759,A -85,B 0,C 180,E1 20943.105,E2 20943.105} C_VEL
LIN {X 0,Y 433.244,Z 411.754,A -85,B 0,C 180,E1 20939.332,E2 20939.332} C_VEL
LIN {X 0,Y 433.24,Z 411.753,A -85,B 0,C 180,E1 20935.478,E2 20935.478} C_VEL
LIN {X 0,Y 433.25,Z 411.752,A -85,B 0,C 180,E1 20931.623,E2 20931.623} C_VEL
LIN {X 0,Y 433.254,Z 411.759,A -85,B 0,C 180,E1 20927.8,E2 20927.8} C_VEL
LIN {X 0,Y 433.253,Z 411.767,A -85,B 0,C 180,E1 20923.941,E2 20923.941} C_VEL
LIN {X 0,Y 433.254,Z 411.76,A -85,B 0,C 180,E1 20920.082,E2 20920.082} C_VEL
LIN {X 0,Y 433.249,Z 411.747,A -85,B 0,C 180,E1 20916.346,E2 20916.346} C_VEL
LIN {X 0,Y 433.247,Z 411.756,A -85,B 0,C 180,E1 20912.529,E2 20912.529} C_VEL
LIN {X 0,Y 433.25,Z 411.768,A -85,B 0,C 180,E1 20908.687,E2 20908.687} C_VEL
LIN {X 0,Y 433.251,Z 411.748,A -85,B 0,C 180,E1 20904.836,E2 20904.836} C_VEL
LIN {X 0,Y 433.249,Z 411.752,A -85,B 0,C 180,E1 20901.102,E2 20901.102} C_VEL
LIN {X 0,Y 433.251,Z 411.765,A -85,B 0,C 180,E1 20897.32,E2 20897.32} C_VEL
LIN {X 0,Y 433.255,Z 411.753,A -85,B 0,C 180,E1 20893.479,E2 20893.479} C_VEL
LIN {X 0,Y 433.248,Z 411.751,A -85,B 0,C 180,E1 20889.699,E2 20889.699} C_VEL
LIN {X 0,Y 433.251,Z 411.766,A -85,B 0,C 180,E1 20885.828,E2 20885.828} C_VEL
LIN {X 0,Y 433.252,Z 411.752,A -85,B 0,C 180,E1 20881.984,E2 20881.984} C_VEL
LIN {X 0,Y 433.245,Z 411.749,A -85,B 0,C 180,E1 20878.281,E2 20878.281} C_VEL
LIN {X 0,Y 433.246,Z 411.766,A -85,B 0,C 180,E1 20874.438,E2 20874.438} C_VEL
LIN {X 0,Y 433.254,Z 411.765,A -85,B 0,C 180,E1 20870.704,E2 20870.704} C_VEL
LIN {X 0,Y 433.253,Z 411.757,A -85,B 0,C 180,E1 20866.883,E2 20866.883} C_VEL
LIN {X 0,Y 433.252,Z 411.751,A -85,B 0,C 180,E1 20863.096,E2 20863.096} C_VEL
LIN {X 0,Y 433.253,Z 411.753,A -85,B 0,C 180,E1 20859.324,E2 20859.324} C_VEL
LIN {X 0,Y 433.241,Z 411.757,A -85,B 0,C 180,E1 20855.6,E2 20855.6} C_VEL
LIN {X 0,Y 433.247,Z 411.756,A -85,B 0,C 180,E1 20851.764,E2 20851.764} C_VEL
LIN {X 0,Y 433.255,Z 411.754,A -85,B 0,C 180,E1 20848.097,E2 20848.097} C_VEL
LIN {X 0,Y 433.254,Z 411.759,A -85,B 0,C 180,E1 20844.277,E2 20844.277} C_VEL
LIN {X 0,Y 433.296,Z 412.034,A -85,B 0,C 180,E1 20841.921,E2 20841.921} C_VEL
LIN {X 0,Y 434.742,Z 415.524,A -85,B 0,C 180,E1 20841.276,E2 20841.276} C_VEL
LIN {X 0,Y 440.067,Z 425.749,A -85,B 0,C 180,E1 20839.473,E2 20839.473} C_VEL
LIN {X 0,Y 448.617,Z 443.499,A -85,B 0,C 180,E1 20836.65,E2 20836.65} C_VEL
LIN {X 0,Y 454.105,Z 455.397,A -85,B 0,C 180,E1 20834.96,E2 20834.96} C_VEL
LIN {X 0,Y 462.793,Z 470.319,A -85,B 0,C 180,E1 20833.685,E2 20833.685} C_VEL
LIN {X 0,Y 465.033,Z 487.507,A -85,B 0,C 180,E1 20833.103,E2 20833.103} C_VEL
LIN {X 0,Y 459.666,Z 707.877,A -85,B 0,C 180,E1 20829.333,E2 20829.333} C_VEL
LIN {X 0,Y 458.284,Z 760.048,A -85,B 0,C 180,E1 20828.42,E2 20828.42} C_VEL
LIN {X 0,Y 456.924,Z 781.837,A -85,B 0,C 180,E1 20827.829,E2 20827.829} C_VEL
LIN {X 0,Y 455.22,Z 802.827,A -85,B 0,C 180,E1 20827.042,E2 20827.042} C_VEL
LIN {X 0,Y 453.271,Z 822.825,A -85,B 0,C 180,E1 20826.086,E2 20826.086} C_VEL
LIN {X 0,Y 450.982,Z 842.771,A -85,B 0,C 180,E1 20824.884,E2 20824.884} C_VEL
LIN {X 0,Y 448.441,Z 862.847,A -85,B 0,C 180,E1 20823.418,E2 20823.418} C_VEL
LIN {X 0,Y 445.931,Z 881.484,A -85,B 0,C 180,E1 20821.799,E2 20821.799} C_VEL
LIN {X 0,Y 443.43,Z 899.27,A -85,B 0,C 180,E1 20819.965,E2 20819.965} C_VEL
LIN {X 0,Y 440.99,Z 916.206,A -85,B 0,C 180,E1 20817.92,E2 20817.92} C_VEL
LIN {X 0,Y 438.75,Z 932.243,A -85,B 0,C 180,E1 20815.659,E2 20815.659} C_VEL
LIN {X 0,Y 436.872,Z 946.434,A -85,B 0,C 180,E1 20813.327,E2 20813.327} C_VEL
LIN {X 0,Y 435.238,Z 959.608,A -85,B 0,C 180,E1 20810.775,E2 20810.775} C_VEL
LIN {X 0,Y 433.928,Z 971.772,A -85,B 0,C 180,E1 20807.987,E2 20807.987} C_VEL
LIN {X 0,Y 433.04,Z 981.698,A -85,B 0,C 180,E1 20805.264,E2 20805.264} C_VEL
LIN {X 0,Y 432.475,Z 989.382,A -85,B 0,C 180,E1 20802.674,E2 20802.674} C_VEL
LIN {X 0,Y 432.133,Z 995.632,A -85,B 0,C 180,E1 20799.996,E2 20799.996} C_VEL
LIN {X 0,Y 431.967,Z 1000.221,A -85,B 0,C 180,E1 20797.317,E2 20797.317} C_VEL
LIN {X 0,Y 431.918,Z 1003.442,A -85,B 0,C 180,E1 20794.517,E2 20794.517} C_VEL
LIN {X 0,Y 431.901,Z 1005.208,A -85,B 0,C 180,E1 20791.727,E2 20791.727} C_VEL
LIN {X 0,Y 431.9,Z 1005.348,A -85,B 0,C 180,E1 20789.074,E2 20789.074} C_VEL
LIN {X 0,Y 431.913,Z 1004.125,A -85,B 0,C 180,E1 20786.287,E2 20786.287} C_VEL
LIN {X 0,Y 431.96,Z 1001.299,A -85,B 0,C 180,E1 20783.491,E2 20783.491} C_VEL
LIN {X 0,Y 432.09,Z 996.912,A -85,B 0,C 180,E1 20780.681,E2 20780.681} C_VEL
LIN {X 0,Y 432.342,Z 991.802,A -85,B 0,C 180,E1 20778.261,E2 20778.261} C_VEL
LIN {X 0,Y 432.822,Z 984.24,A -85,B 0,C 180,E1 20775.556,E2 20775.556} C_VEL
LIN {X 0,Y 433.566,Z 975.47,A -85,B 0,C 180,E1 20772.973,E2 20772.973} C_VEL
LIN {X 0,Y 434.636,Z 964.781,A -85,B 0,C 180,E1 20770.378,E2 20770.378} C_VEL
LIN {X 0,Y 436.093,Z 952.152,A -85,B 0,C 180,E1 20767.775,E2 20767.775} C_VEL
LIN {X 0,Y 437.869,Z 938.332,A -85,B 0,C 180,E1 20765.342,E2 20765.342} C_VEL
LIN {X 0,Y 439.938,Z 922.928,A -85,B 0,C 180,E1 20763.041,E2 20763.041} C_VEL
LIN {X 0,Y 442.239,Z 906.365,A -85,B 0,C 180,E1 20760.92,E2 20760.92} C_VEL
LIN {X 0,Y 444.685,Z 889.027,A -85,B 0,C 180,E1 20759.014,E2 20759.014} C_VEL
LIN {X 0,Y 447.14,Z 870.889,A -85,B 0,C 180,E1 20757.319,E2 20757.319} C_VEL
LIN {X 0,Y 449.534,Z 852.054,A -85,B 0,C 180,E1 20755.833,E2 20755.833} C_VEL
LIN {X 0,Y 451.976,Z 831.737,A -85,B 0,C 180,E1 20754.497,E2 20754.497} C_VEL
LIN {X 0,Y 454.071,Z 811.48,A -85,B 0,C 180,E1 20753.414,E2 20753.414} C_VEL
LIN {X 0,Y 455.926,Z 790.213,A -85,B 0,C 180,E1 20752.526,E2 20752.526} C_VEL
LIN {X 0,Y 457.497,Z 768.005,A -85,B 0,C 180,E1 20751.838,E2 20751.838} C_VEL
LIN {X 0,Y 458.477,Z 745.652,A -85,B 0,C 180,E1 20751.364,E2 20751.364} C_VEL
LIN {X 0,Y 463.762,Z 520.257,A -85,B 0,C 180,E1 20747.531,E2 20747.531} C_VEL
LIN {X 0,Y 464.463,Z 485.151,A -85,B 0,C 180,E1 20746.901,E2 20746.901} C_VEL
LIN {X 0,Y 462.113,Z 469.112,A -85,B 0,C 180,E1 20746.319,E2 20746.319} C_VEL
LIN {X 0,Y 453.611,Z 454.586,A -85,B 0,C 180,E1 20745.036,E2 20745.036} C_VEL
LIN {X 0,Y 445.912,Z 437.385,A -85,B 0,C 180,E1 20742.448,E2 20742.448} C_VEL
LIN {X 0,Y 439.573,Z 424.624,A -85,B 0,C 180,E1 20740.239,E2 20740.239} C_VEL
LIN {X 0,Y 437.184,Z 420.092,A -85,B 0,C 180,E1 20739.381,E2 20739.381} C_VEL
LIN {X 0,Y 434.92,Z 415.766,A -85,B 0,C 180,E1 20738.536,E2 20738.536} C_VEL
LIN {X 0,Y 433.283,Z 412.006,A -85,B 0,C 180,E1 20737.751,E2 20737.751} C_VEL
LIN {X 0,Y 433.252,Z 411.762,A -85,B 0,C 180,E1 20734.063,E2 20734.063} C_VEL
LIN {X 0,Y 433.224,Z 411.773,A -85,B 0,C 180,E1 20730.334,E2 20730.334} C_VEL
LIN {X 0,Y 433.198,Z 411.764,A -85,B 0,C 180,E1 20726.728,E2 20726.728} C_VEL
LIN {X 0,Y 433.198,Z 411.772,A -85,B 0,C 180,E1 20722.95,E2 20722.95} C_VEL
LIN {X 0,Y 433.219,Z 411.773,A -85,B 0,C 180,E1 20719.286,E2 20719.286} C_VEL
LIN {X 0,Y 433.238,Z 411.764,A -85,B 0,C 180,E1 20715.528,E2 20715.528} C_VEL
LIN {X 0,Y 433.212,Z 411.764,A -85,B 0,C 180,E1 20711.718,E2 20711.718} C_VEL
LIN {X 0,Y 433.192,Z 411.763,A -85,B 0,C 180,E1 20708.068,E2 20708.068} C_VEL
LIN {X 0,Y 433.195,Z 411.77,A -85,B 0,C 180,E1 20704.368,E2 20704.368} C_VEL
LIN {X 0,Y 433.217,Z 411.773,A -85,B 0,C 180,E1 20700.661,E2 20700.661} C_VEL
LIN {X 0,Y 433.25,Z 411.762,A -85,B 0,C 180,E1 20696.957,E2 20696.957} C_VEL
LIN {X 0,Y 433.258,Z 411.761,A -85,B 0,C 180,E1 20693.107,E2 20693.107} C_VEL
LIN {X 0,Y 433.239,Z 411.768,A -85,B 0,C 180,E1 20689.36,E2 20689.36} C_VEL
LIN {X 0,Y 433.229,Z 411.771,A -85,B 0,C 180,E1 20685.566,E2 20685.566} C_VEL
LIN {X 0,Y 433.316,Z 412.165,A -85,B 0,C 180,E1 20684.457,E2 20684.457} C_VEL
LIN {X 0,Y 434.807,Z 415.637,A -85,B 0,C 180,E1 20683.707,E2 20683.707} C_VEL
LIN {X 0,Y 438.058,Z 422.247,A -85,B 0,C 180,E1 20682.327,E2 20682.327} C_VEL
LIN {X 0,Y 443.527,Z 433.778,A -85,B 0,C 180,E1 20680.098,E2 20680.098} C_VEL
LIN {X 0,Y 450.472,Z 450.122,A -85,B 0,C 180,E1 20677.281,E2 20677.281} C_VEL
LIN {X 0,Y 452.048,Z 453.749,A -85,B 0,C 180,E1 20676.762,E2 20676.762} C_VEL
LIN {X 0,Y 458.914,Z 465.544,A -85,B 0,C 180,E1 20675.691,E2 20675.691} C_VEL
LIN {X 0,Y 461.993,Z 484.678,A -85,B 0,C 180,E1 20674.928,E2 20674.928} C_VEL
LIN {X 0,Y 454.947,Z 720.021,A -85,B 0,C 180,E1 20670.722,E2 20670.722} C_VEL
LIN {X 0,Y 453.743,Z 741.028,A -85,B 0,C 180,E1 20670.114,E2 20670.114} C_VEL
LIN {X 0,Y 452.225,Z 760.639,A -85,B 0,C 180,E1 20669.316,E2 20669.316} C_VEL
LIN {X 0,Y 450.436,Z 779.471,A -85,B 0,C 180,E1 20668.326,E2 20668.326} C_VEL
LIN {X 0,Y 448.338,Z 798.245,A -85,B 0,C 180,E1 20667.095,E2 20667.095} C_VEL
LIN {X 0,Y 446.121,Z 816.007,A -85,B 0,C 180,E1 20665.671,E2 20665.671} C_VEL
LIN {X 0,Y 443.704,Z 833.464,A -85,B 0,C 180,E1 20663.974,E2 20663.974} C_VEL
LIN {X 0,Y 441.401,Z 849.267,A -85,B 0,C 180,E1 20662.13,E2 20662.13} C_VEL
LIN {X 0,Y 439.234,Z 863.965,A -85,B 0,C 180,E1 20660.091,E2 20660.091} C_VEL
LIN {X 0,Y 438.103,Z 871.655,A -85,B 0,C 180,E1 20658.872,E2 20658.872} C_VEL
LIN {X 0,Y 436.483,Z 876.534,A -85,B 0,C 180,E1 20658.105,E2 20658.105} C_VEL
LIN {X 0,Y 429.173,Z 888.456,A -85,B 0,C 180,E1 20656.181,E2 20656.181} C_VEL
LIN {X 0,Y 427.652,Z 892.536,A -85,B 0,C 180,E1 20655.33,E2 20655.33} C_VEL
LIN {X 0,Y 426.301,Z 902.675,A -85,B 0,C 180,E1 20652.767,E2 20652.767} C_VEL
LIN {X 0,Y 425.32,Z 911.256,A -85,B 0,C 180,E1 20650.095,E2 20650.095} C_VEL
LIN {X 0,Y 424.689,Z 918.102,A -85,B 0,C 180,E1 20647.398,E2 20647.398} C_VEL
LIN {X 0,Y 424.333,Z 923.308,A -85,B 0,C 180,E1 20644.678,E2 20644.678} C_VEL
LIN {X 0,Y 424.156,Z 926.925,A -85,B 0,C 180,E1 20641.868,E2 20641.868} C_VEL
LIN {X 0,Y 424.091,Z 928.825,A -85,B 0,C 180,E1 20639.207,E2 20639.207} C_VEL
LIN {X 0,Y 424.072,Z 929.279,A -85,B 0,C 180,E1 20636.369,E2 20636.369} C_VEL
LIN {X 0,Y 424.093,Z 928.168,A -85,B 0,C 180,E1 20633.624,E2 20633.624} C_VEL
LIN {X 0,Y 424.204,Z 925.431,A -85,B 0,C 180,E1 20630.845,E2 20630.845} C_VEL
LIN {X 0,Y 424.427,Z 921.083,A -85,B 0,C 180,E1 20628.114,E2 20628.114} C_VEL
LIN {X 0,Y 424.856,Z 915.179,A -85,B 0,C 180,E1 20625.419,E2 20625.419} C_VEL
LIN {X 0,Y 425.647,Z 907.18,A -85,B 0,C 180,E1 20622.615,E2 20622.615} C_VEL
LIN {X 0,Y 426.764,Z 897.753,A -85,B 0,C 180,E1 20619.981,E2 20619.981} C_VEL
LIN {X 0,Y 428.221,Z 886.995,A -85,B 0,C 180,E1 20617.51,E2 20617.51} C_VEL
LIN {X 0,Y 430.102,Z 874.146,A -85,B 0,C 180,E1 20615.065,E2 20615.065} C_VEL
LIN {X 0,Y 432.291,Z 859.696,A -85,B 0,C 180,E1 20612.781,E2 20612.781} C_VEL
LIN {X 0,Y 434.574,Z 844.608,A -85,B 0,C 180,E1 20610.788,E2 20610.788} C_VEL
LIN {X 0,Y 436.928,Z 828.64,A -85,B 0,C 180,E1 20609.014,E2 20609.014} C_VEL
LIN {X 0,Y 439.418,Z 810.492,A -85,B 0,C 180,E1 20607.33,E2 20607.33} C_VEL
LIN {X 0,Y 441.747,Z 792.16,A -85,B 0,C 180,E1 20605.934,E2 20605.934} C_VEL
LIN {X 0,Y 443.815,Z 773.382,A -85,B 0,C 180,E1 20604.769,E2 20604.769} C_VEL
LIN {X 0,Y 445.68,Z 753.109,A -85,B 0,C 180,E1 20603.783,E2 20603.783} C_VEL
LIN {X 0,Y 447.115,Z 732.732,A -85,B 0,C 180,E1 20603.05,E2 20603.05} C_VEL
LIN {X 0,Y 448.095,Z 712.097,A -85,B 0,C 180,E1 20602.537,E2 20602.537} C_VEL
LIN {X 0,Y 454.518,Z 484.603,A -85,B 0,C 180,E1 20598.518,E2 20598.518} C_VEL
LIN {X 0,Y 451.347,Z 467.247,A -85,B 0,C 180,E1 20597.809,E2 20597.809} C_VEL
LIN {X 0,Y 442.641,Z 452.424,A -85,B 0,C 180,E1 20596.477,E2 20596.477} C_VEL
LIN {X 0,Y 435.726,Z 435.822,A -85,B 0,C 180,E1 20593.74,E2 20593.74} C_VEL
LIN {X 0,Y 429.123,Z 421.131,A -85,B 0,C 180,E1 20591.083,E2 20591.083} C_VEL
LIN {X 0,Y 425.402,Z 413.314,A -85,B 0,C 180,E1 20589.534,E2 20589.534} C_VEL
LIN {X 0,Y 425.314,Z 412.724,A -85,B 0,C 180,E1 20589.061,E2 20589.061} C_VEL
LIN {X 0,Y 425.311,Z 412.73,A -85,B 0,C 180,E1 20585.26,E2 20585.26} C_VEL
LIN {X 0,Y 425.307,Z 412.752,A -85,B 0,C 180,E1 20581.493,E2 20581.493} C_VEL
LIN {X 0,Y 425.304,Z 412.756,A -85,B 0,C 180,E1 20577.564,E2 20577.564} C_VEL
LIN {X 0,Y 425.309,Z 412.754,A -85,B 0,C 180,E1 20573.668,E2 20573.668} C_VEL
LIN {X 0,Y 425.318,Z 412.745,A -85,B 0,C 180,E1 20569.821,E2 20569.821} C_VEL
LIN {X 0,Y 425.313,Z 412.737,A -85,B 0,C 180,E1 20565.902,E2 20565.902} C_VEL
LIN {X 0,Y 425.311,Z 412.737,A -85,B 0,C 180,E1 20562.02,E2 20562.02} C_VEL
LIN {X 0,Y 425.319,Z 412.751,A -85,B 0,C 180,E1 20558.191,E2 20558.191} C_VEL
LIN {X 0,Y 425.312,Z 412.755,A -85,B 0,C 180,E1 20554.348,E2 20554.348} C_VEL
LIN {X 0,Y 425.308,Z 412.74,A -85,B 0,C 180,E1 20550.518,E2 20550.518} C_VEL
LIN {X 0,Y 425.311,Z 412.736,A -85,B 0,C 180,E1 20546.681,E2 20546.681} C_VEL
LIN {X 0,Y 425.319,Z 412.757,A -85,B 0,C 180,E1 20542.824,E2 20542.824} C_VEL
LIN {X 0,Y 425.31,Z 412.74,A -85,B 0,C 180,E1 20538.931,E2 20538.931} C_VEL
LIN {X 0,Y 425.308,Z 412.738,A -85,B 0,C 180,E1 20535.127,E2 20535.127} C_VEL
LIN {X 0,Y 425.315,Z 412.754,A -85,B 0,C 180,E1 20531.252,E2 20531.252} C_VEL
